// TIA Portal V18 program export: 1 tag tables, 0 data types, 4 data blocks, 9 code blocks (in call order from the OBs), 0 instance data blocks

VAR_GLOBAL   // PLC tag table "PLC_Tags"
   Nut_Khoi_Dong AT %I0.0 : Bool;   // Nút khởi động vật lý
   Nut_Khoi_Dong_HMI AT %M110.0 : Bool;   // Tín hiệu mô phỏng/HMI song song cho Nút khởi động vật lý
   Nut_Khoi_Dong_HMI_Gated AT %M320.0 : Bool;   // Tín hiệu HMI đã qua xử lý chế độ cho Nút khởi động vật lý
   Nut_Khoi_Dong_Eff AT %M320.1 : Bool;   // Tín hiệu thực tế/mô phỏng hiệu dụng cho Nút khởi động vật lý
   Nut_Dung AT %I0.1 : Bool;   // Nút dừng vật lý
   Nut_Dung_HMI AT %M110.1 : Bool;   // Tín hiệu mô phỏng/HMI song song cho Nút dừng vật lý
   Nut_Dung_HMI_Gated AT %M320.2 : Bool;   // Tín hiệu HMI đã qua xử lý chế độ cho Nút dừng vật lý
   Nut_Dung_Eff AT %M320.3 : Bool;   // Tín hiệu thực tế/mô phỏng hiệu dụng cho Nút dừng vật lý
   Nut_Reset AT %I0.2 : Bool;   // Nút reset lỗi vật lý
   Nut_Reset_HMI AT %M110.2 : Bool;   // Tín hiệu mô phỏng/HMI song song cho Nút reset lỗi vật lý
   Nut_Reset_HMI_Gated AT %M320.4 : Bool;   // Tín hiệu HMI đã qua xử lý chế độ cho Nút reset lỗi vật lý
   Nut_Reset_Eff AT %M320.5 : Bool;   // Tín hiệu thực tế/mô phỏng hiệu dụng cho Nút reset lỗi vật lý
   Nut_EStop AT %I0.3 : Bool;   // Nút dừng khẩn vật lý
   Nut_EStop_HMI AT %M110.3 : Bool;   // Tín hiệu mô phỏng/HMI song song cho Nút dừng khẩn vật lý
   Nut_EStop_HMI_Gated AT %M320.6 : Bool;   // Tín hiệu HMI đã qua xử lý chế độ cho Nút dừng khẩn vật lý
   Nut_EStop_Eff AT %M320.7 : Bool;   // Tín hiệu thực tế/mô phỏng hiệu dụng cho Nút dừng khẩn vật lý
   FT3200_Bon1 AT %ID100 : Real;   // Cảm biến lưu lượng nước dosing vào Bồn 1
   FT3200_Bon1_HMI AT %MD700 : Real;   // Giá trị mô phỏng/HMI song song cho Cảm biến lưu lượng nước dosing vào Bồn 1
   FT3200_Bon1_Use_HMI AT %M420.0 : Bool;   // Chọn chế độ mô phỏng HMI cho Cảm biến lưu lượng nước dosing vào Bồn 1
   FT3200_Bon1_Sim_Req AT %M321.0 : Bool;   // Yêu cầu mô phỏng cảm biến cho Cảm biến lưu lượng nước dosing vào Bồn 1
   FT3200_Bon1_Sim_Active AT %M321.1 : Bool;   // Mô phỏng cảm biến đang hoạt động cho Cảm biến lưu lượng nước dosing vào Bồn 1
   FT3200_Bon1_Eff AT %MD704 : Real;   // Giá trị thực tế/mô phỏng hiệu dụng cho Cảm biến lưu lượng nước dosing vào Bồn 1
   FQ3200_Bon1 AT %ID104 : Real;   // Bộ đếm lưu lượng tích lũy Bồn 1
   FQ3200_Bon1_HMI AT %MD708 : Real;   // Giá trị mô phỏng/HMI song song cho Bộ đếm lưu lượng tích lũy Bồn 1
   FQ3200_Bon1_Use_HMI AT %M420.1 : Bool;   // Chọn chế độ mô phỏng HMI cho Bộ đếm lưu lượng tích lũy Bồn 1
   FQ3200_Bon1_Sim_Req AT %M321.2 : Bool;   // Yêu cầu mô phỏng cảm biến cho Bộ đếm lưu lượng tích lũy Bồn 1
   FQ3200_Bon1_Sim_Active AT %M321.3 : Bool;   // Mô phỏng cảm biến đang hoạt động cho Bộ đếm lưu lượng tích lũy Bồn 1
   FQ3200_Bon1_Eff AT %MD712 : Real;   // Giá trị thực tế/mô phỏng hiệu dụng cho Bộ đếm lưu lượng tích lũy Bồn 1
   LS3202_Bon1_Cao AT %I0.4 : Bool;   // Cảm biến mức cao Bồn 1
   LS3202_Bon1_Cao_HMI AT %M110.4 : Bool;   // Tín hiệu mô phỏng/HMI song song cho Cảm biến mức cao Bồn 1
   LS3202_Bon1_Cao_HMI_Gated AT %M321.4 : Bool;   // Tín hiệu HMI đã qua xử lý chế độ cho Cảm biến mức cao Bồn 1
   LS3202_Bon1_Cao_Eff AT %M321.5 : Bool;   // Tín hiệu thực tế/mô phỏng hiệu dụng cho Cảm biến mức cao Bồn 1
   LT3203_Bon1 AT %ID108 : Real;   // Cảm biến mức liên tục Bồn 1
   LT3203_Bon1_HMI AT %MD716 : Real;   // Giá trị mô phỏng/HMI song song cho Cảm biến mức liên tục Bồn 1
   LT3203_Bon1_Use_HMI AT %M420.2 : Bool;   // Chọn chế độ mô phỏng HMI cho Cảm biến mức liên tục Bồn 1
   LT3203_Bon1_Sim_Req AT %M321.6 : Bool;   // Yêu cầu mô phỏng cảm biến cho Cảm biến mức liên tục Bồn 1
   LT3203_Bon1_Sim_Active AT %M321.7 : Bool;   // Mô phỏng cảm biến đang hoạt động cho Cảm biến mức liên tục Bồn 1
   LT3203_Bon1_Eff AT %MD720 : Real;   // Giá trị thực tế/mô phỏng hiệu dụng cho Cảm biến mức liên tục Bồn 1
   TT3204_Bon1 AT %ID112 : Real;   // Cảm biến nhiệt độ Bồn 1
   TT3204_Bon1_HMI AT %MD724 : Real;   // Giá trị mô phỏng/HMI song song cho Cảm biến nhiệt độ Bồn 1
   TT3204_Bon1_Use_HMI AT %M420.3 : Bool;   // Chọn chế độ mô phỏng HMI cho Cảm biến nhiệt độ Bồn 1
   TT3204_Bon1_Sim_Req AT %M322.0 : Bool;   // Yêu cầu mô phỏng cảm biến cho Cảm biến nhiệt độ Bồn 1
   TT3204_Bon1_Sim_Active AT %M322.1 : Bool;   // Mô phỏng cảm biến đang hoạt động cho Cảm biến nhiệt độ Bồn 1
   TT3204_Bon1_Eff AT %MD728 : Real;   // Giá trị thực tế/mô phỏng hiệu dụng cho Cảm biến nhiệt độ Bồn 1
   FT3205_Bon2 AT %ID116 : Real;   // Cảm biến lưu lượng nước dosing vào Bồn 2
   FT3205_Bon2_HMI AT %MD732 : Real;   // Giá trị mô phỏng/HMI song song cho Cảm biến lưu lượng nước dosing vào Bồn 2
   FT3205_Bon2_Use_HMI AT %M420.4 : Bool;   // Chọn chế độ mô phỏng HMI cho Cảm biến lưu lượng nước dosing vào Bồn 2
   FT3205_Bon2_Sim_Req AT %M322.2 : Bool;   // Yêu cầu mô phỏng cảm biến cho Cảm biến lưu lượng nước dosing vào Bồn 2
   FT3205_Bon2_Sim_Active AT %M322.3 : Bool;   // Mô phỏng cảm biến đang hoạt động cho Cảm biến lưu lượng nước dosing vào Bồn 2
   FT3205_Bon2_Eff AT %MD736 : Real;   // Giá trị thực tế/mô phỏng hiệu dụng cho Cảm biến lưu lượng nước dosing vào Bồn 2
   FQ3205_Bon2 AT %ID120 : Real;   // Bộ đếm lưu lượng tích lũy Bồn 2
   FQ3205_Bon2_HMI AT %MD740 : Real;   // Giá trị mô phỏng/HMI song song cho Bộ đếm lưu lượng tích lũy Bồn 2
   FQ3205_Bon2_Use_HMI AT %M420.5 : Bool;   // Chọn chế độ mô phỏng HMI cho Bộ đếm lưu lượng tích lũy Bồn 2
   FQ3205_Bon2_Sim_Req AT %M322.4 : Bool;   // Yêu cầu mô phỏng cảm biến cho Bộ đếm lưu lượng tích lũy Bồn 2
   FQ3205_Bon2_Sim_Active AT %M322.5 : Bool;   // Mô phỏng cảm biến đang hoạt động cho Bộ đếm lưu lượng tích lũy Bồn 2
   FQ3205_Bon2_Eff AT %MD744 : Real;   // Giá trị thực tế/mô phỏng hiệu dụng cho Bộ đếm lưu lượng tích lũy Bồn 2
   LT3209_Bon2 AT %ID124 : Real;   // Cảm biến mức liên tục Bồn 2
   LT3209_Bon2_HMI AT %MD748 : Real;   // Giá trị mô phỏng/HMI song song cho Cảm biến mức liên tục Bồn 2
   LT3209_Bon2_Use_HMI AT %M420.6 : Bool;   // Chọn chế độ mô phỏng HMI cho Cảm biến mức liên tục Bồn 2
   LT3209_Bon2_Sim_Req AT %M322.6 : Bool;   // Yêu cầu mô phỏng cảm biến cho Cảm biến mức liên tục Bồn 2
   LT3209_Bon2_Sim_Active AT %M322.7 : Bool;   // Mô phỏng cảm biến đang hoạt động cho Cảm biến mức liên tục Bồn 2
   LT3209_Bon2_Eff AT %MD752 : Real;   // Giá trị thực tế/mô phỏng hiệu dụng cho Cảm biến mức liên tục Bồn 2
   TT3208_Bon2 AT %ID128 : Real;   // Cảm biến nhiệt độ Bồn 2
   TT3208_Bon2_HMI AT %MD756 : Real;   // Giá trị mô phỏng/HMI song song cho Cảm biến nhiệt độ Bồn 2
   TT3208_Bon2_Use_HMI AT %M420.7 : Bool;   // Chọn chế độ mô phỏng HMI cho Cảm biến nhiệt độ Bồn 2
   TT3208_Bon2_Sim_Req AT %M323.0 : Bool;   // Yêu cầu mô phỏng cảm biến cho Cảm biến nhiệt độ Bồn 2
   TT3208_Bon2_Sim_Active AT %M323.1 : Bool;   // Mô phỏng cảm biến đang hoạt động cho Cảm biến nhiệt độ Bồn 2
   TT3208_Bon2_Eff AT %MD760 : Real;   // Giá trị thực tế/mô phỏng hiệu dụng cho Cảm biến nhiệt độ Bồn 2
   VFD_Bon2_Contactor AT %Q0.0 : Bool;   // Contactor cấp nguồn/cho phép VFD Bồn 2
   VFD_Bon2_Contactor_M AT %M220.0 : Bool;   // Tag gương phản hồi HMI cho Contactor cấp nguồn/cho phép VFD Bồn 2
   CV3201_Nuoc_Bon1 AT %QD100 : Real;   // Van tuyến tính cấp nước Bồn 1
   CV3201_Nuoc_Bon1_M AT %MD1200 : Real;   // Tag gương phản hồi HMI cho Van tuyến tính cấp nước Bồn 1
   AGTR3260_Khuay_Bon1 AT %Q0.1 : Bool;   // Động cơ khuấy Bồn 1
   AGTR3260_Khuay_Bon1_M AT %M220.1 : Bool;   // Tag gương phản hồi HMI cho Động cơ khuấy Bồn 1
   AGTR3260_Toc_Do_AO AT %QD104 : Real;   // Tín hiệu tốc độ khuấy Bồn 1
   AGTR3260_Toc_Do_AO_M AT %MD1204 : Real;   // Tag gương phản hồi HMI cho Tín hiệu tốc độ khuấy Bồn 1
   V3232_Xa_Bon1 AT %Q0.2 : Bool;   // Van xả đáy Bồn 1 số 1
   V3232_Xa_Bon1_M AT %M220.2 : Bool;   // Tag gương phản hồi HMI cho Van xả đáy Bồn 1 số 1
   V3233_Xa_Bon1 AT %Q0.3 : Bool;   // Van xả đáy Bồn 1 số 2
   V3233_Xa_Bon1_M AT %M220.3 : Bool;   // Tag gương phản hồi HMI cho Van xả đáy Bồn 1 số 2
   V3234_Xa_Bon1 AT %Q0.4 : Bool;   // Van xả đáy Bồn 1 số 3
   V3234_Xa_Bon1_M AT %M220.4 : Bool;   // Tag gương phản hồi HMI cho Van xả đáy Bồn 1 số 3
   V3235_Nuoc_Bon2 AT %Q0.5 : Bool;   // Van on/off cấp nước Bồn 2
   V3235_Nuoc_Bon2_M AT %M220.5 : Bool;   // Tag gương phản hồi HMI cho Van on/off cấp nước Bồn 2
   CV3206_Hoi_Bon2 AT %QD108 : Real;   // Van hơi/nhiệt Bồn 2 ở chế độ cho phép
   CV3206_Hoi_Bon2_M AT %MD1208 : Real;   // Tag gương phản hồi HMI cho Van hơi/nhiệt Bồn 2 ở chế độ cho phép
   VFD_Bon2_Dummy_Run_Physical AT %Q0.6 : Bool;   // Dummy RUN physical output VFD Bồn 2
   VFD_Bon2_Dummy_Run_Physical_M AT %M220.6 : Bool;   // Tag gương phản hồi HMI cho Dummy RUN physical output VFD Bồn 2
   VFD_Bon2_Dummy_Reverse_Physical AT %Q0.7 : Bool;   // Dummy Reverse physical output VFD Bồn 2
   VFD_Bon2_Dummy_Reverse_Physical_M AT %M220.7 : Bool;   // Tag gương phản hồi HMI cho Dummy Reverse physical output VFD Bồn 2
   VFD_Bon2_Dummy_Speed_Physical AT %QD112 : Real;   // Dummy Speed physical output VFD Bồn 2
   VFD_Bon2_Dummy_Speed_Physical_M AT %MD1212 : Real;   // Tag gương phản hồi HMI cho Dummy Speed physical output VFD Bồn 2
   V3237_Xa_Bon2 AT %Q1.0 : Bool;   // Van xả đáy Bồn 2 số 1
   V3237_Xa_Bon2_M AT %M221.0 : Bool;   // Tag gương phản hồi HMI cho Van xả đáy Bồn 2 số 1
   V3238_Xa_Bon2 AT %Q1.1 : Bool;   // Van xả đáy Bồn 2 số 2
   V3238_Xa_Bon2_M AT %M221.1 : Bool;   // Tag gương phản hồi HMI cho Van xả đáy Bồn 2 số 2
   V3239_Xa_Bon2 AT %Q1.2 : Bool;   // Van xả đáy Bồn 2 số 3
   V3239_Xa_Bon2_M AT %M221.2 : Bool;   // Tag gương phản hồi HMI cho Van xả đáy Bồn 2 số 3
   Pump3264_Chuyen_Nhanh1 AT %Q1.3 : Bool;   // Bơm chuyển dung dịch Nhánh 1 xuống bồn chứa
   Pump3264_Chuyen_Nhanh1_M AT %M221.3 : Bool;   // Tag gương phản hồi HMI cho Bơm chuyển dung dịch Nhánh 1 xuống bồn chứa
   LT3302_BonChua1 AT %ID164 : Real;   // Cảm biến mức liên tục Bồn chứa 01
   LT3302_BonChua1_HMI AT %MD828 : Real;   // Giá trị mô phỏng/HMI song song cho Cảm biến mức liên tục Bồn chứa 01
   LT3302_BonChua1_Use_HMI AT %M422.0 : Bool;   // Chọn chế độ mô phỏng HMI cho Cảm biến mức liên tục Bồn chứa 01
   LT3302_BonChua1_Sim_Req AT %M325.4 : Bool;   // Yêu cầu mô phỏng cảm biến cho Cảm biến mức liên tục Bồn chứa 01
   LT3302_BonChua1_Sim_Active AT %M325.5 : Bool;   // Mô phỏng cảm biến đang hoạt động cho Cảm biến mức liên tục Bồn chứa 01
   LT3302_BonChua1_Eff AT %MD832 : Real;   // Giá trị thực tế/mô phỏng hiệu dụng cho Cảm biến mức liên tục Bồn chứa 01
   TT3301_BonChua1 AT %ID168 : Real;   // Cảm biến nhiệt độ Bồn chứa 01
   TT3301_BonChua1_HMI AT %MD836 : Real;   // Giá trị mô phỏng/HMI song song cho Cảm biến nhiệt độ Bồn chứa 01
   TT3301_BonChua1_Use_HMI AT %M422.1 : Bool;   // Chọn chế độ mô phỏng HMI cho Cảm biến nhiệt độ Bồn chứa 01
   TT3301_BonChua1_Sim_Req AT %M325.6 : Bool;   // Yêu cầu mô phỏng cảm biến cho Cảm biến nhiệt độ Bồn chứa 01
   TT3301_BonChua1_Sim_Active AT %M325.7 : Bool;   // Mô phỏng cảm biến đang hoạt động cho Cảm biến nhiệt độ Bồn chứa 01
   TT3301_BonChua1_Eff AT %MD840 : Real;   // Giá trị thực tế/mô phỏng hiệu dụng cho Cảm biến nhiệt độ Bồn chứa 01
   TT3303_TraoDoiNhiet AT %ID172 : Real;   // Cảm biến nhiệt độ bộ trao đổi nhiệt
   TT3303_TraoDoiNhiet_HMI AT %MD844 : Real;   // Giá trị mô phỏng/HMI song song cho Cảm biến nhiệt độ bộ trao đổi nhiệt
   TT3303_TraoDoiNhiet_Use_HMI AT %M422.2 : Bool;   // Chọn chế độ mô phỏng HMI cho Cảm biến nhiệt độ bộ trao đổi nhiệt
   TT3303_TraoDoiNhiet_Sim_Req AT %M326.0 : Bool;   // Yêu cầu mô phỏng cảm biến cho Cảm biến nhiệt độ bộ trao đổi nhiệt
   TT3303_TraoDoiNhiet_Sim_Active AT %M326.1 : Bool;   // Mô phỏng cảm biến đang hoạt động cho Cảm biến nhiệt độ bộ trao đổi nhiệt
   TT3303_TraoDoiNhiet_Eff AT %MD848 : Real;   // Giá trị thực tế/mô phỏng hiệu dụng cho Cảm biến nhiệt độ bộ trao đổi nhiệt
   LT3307_BonChua2 AT %ID176 : Real;   // Cảm biến mức liên tục Bồn chứa 02
   LT3307_BonChua2_HMI AT %MD852 : Real;   // Giá trị mô phỏng/HMI song song cho Cảm biến mức liên tục Bồn chứa 02
   LT3307_BonChua2_Use_HMI AT %M422.3 : Bool;   // Chọn chế độ mô phỏng HMI cho Cảm biến mức liên tục Bồn chứa 02
   LT3307_BonChua2_Sim_Req AT %M326.2 : Bool;   // Yêu cầu mô phỏng cảm biến cho Cảm biến mức liên tục Bồn chứa 02
   LT3307_BonChua2_Sim_Active AT %M326.3 : Bool;   // Mô phỏng cảm biến đang hoạt động cho Cảm biến mức liên tục Bồn chứa 02
   LT3307_BonChua2_Eff AT %MD856 : Real;   // Giá trị thực tế/mô phỏng hiệu dụng cho Cảm biến mức liên tục Bồn chứa 02
   TT3306_BonChua2 AT %ID180 : Real;   // Cảm biến nhiệt độ Bồn chứa 02
   TT3306_BonChua2_HMI AT %MD860 : Real;   // Giá trị mô phỏng/HMI song song cho Cảm biến nhiệt độ Bồn chứa 02
   TT3306_BonChua2_Use_HMI AT %M422.4 : Bool;   // Chọn chế độ mô phỏng HMI cho Cảm biến nhiệt độ Bồn chứa 02
   TT3306_BonChua2_Sim_Req AT %M326.4 : Bool;   // Yêu cầu mô phỏng cảm biến cho Cảm biến nhiệt độ Bồn chứa 02
   TT3306_BonChua2_Sim_Active AT %M326.5 : Bool;   // Mô phỏng cảm biến đang hoạt động cho Cảm biến nhiệt độ Bồn chứa 02
   TT3306_BonChua2_Eff AT %MD864 : Real;   // Giá trị thực tế/mô phỏng hiệu dụng cho Cảm biến nhiệt độ Bồn chứa 02
   PI3308_Truoc_Filter AT %ID184 : Real;   // Cảm biến áp suất trước màng lọc
   PI3308_Truoc_Filter_HMI AT %MD868 : Real;   // Giá trị mô phỏng/HMI song song cho Cảm biến áp suất trước màng lọc
   PI3308_Truoc_Filter_Use_HMI AT %M422.5 : Bool;   // Chọn chế độ mô phỏng HMI cho Cảm biến áp suất trước màng lọc
   PI3308_Truoc_Filter_Sim_Req AT %M326.6 : Bool;   // Yêu cầu mô phỏng cảm biến cho Cảm biến áp suất trước màng lọc
   PI3308_Truoc_Filter_Sim_Active AT %M326.7 : Bool;   // Mô phỏng cảm biến đang hoạt động cho Cảm biến áp suất trước màng lọc
   PI3308_Truoc_Filter_Eff AT %MD872 : Real;   // Giá trị thực tế/mô phỏng hiệu dụng cho Cảm biến áp suất trước màng lọc
   FT3309_Xa_Thanh_Pham AT %ID188 : Real;   // Cảm biến lưu lượng xả thành phẩm
   FT3309_Xa_Thanh_Pham_HMI AT %MD876 : Real;   // Giá trị mô phỏng/HMI song song cho Cảm biến lưu lượng xả thành phẩm
   FT3309_Xa_Thanh_Pham_Use_HMI AT %M422.6 : Bool;   // Chọn chế độ mô phỏng HMI cho Cảm biến lưu lượng xả thành phẩm
   FT3309_Xa_Thanh_Pham_Sim_Req AT %M327.0 : Bool;   // Yêu cầu mô phỏng cảm biến cho Cảm biến lưu lượng xả thành phẩm
   FT3309_Xa_Thanh_Pham_Sim_Active AT %M327.1 : Bool;   // Mô phỏng cảm biến đang hoạt động cho Cảm biến lưu lượng xả thành phẩm
   FT3309_Xa_Thanh_Pham_Eff AT %MD880 : Real;   // Giá trị thực tế/mô phỏng hiệu dụng cho Cảm biến lưu lượng xả thành phẩm
   LSH3310_Pheu_Cao AT %I0.6 : Bool;   // Cảm biến mức cao phễu chiết rót
   LSH3310_Pheu_Cao_HMI AT %M110.6 : Bool;   // Tín hiệu mô phỏng/HMI song song cho Cảm biến mức cao phễu chiết rót
   LSH3310_Pheu_Cao_HMI_Gated AT %M327.2 : Bool;   // Tín hiệu HMI đã qua xử lý chế độ cho Cảm biến mức cao phễu chiết rót
   LSH3310_Pheu_Cao_Eff AT %M327.3 : Bool;   // Tín hiệu thực tế/mô phỏng hiệu dụng cho Cảm biến mức cao phễu chiết rót
   LSL3311_Pheu_Thap AT %I0.7 : Bool;   // Cảm biến mức thấp phễu chiết rót
   LSL3311_Pheu_Thap_HMI AT %M110.7 : Bool;   // Tín hiệu mô phỏng/HMI song song cho Cảm biến mức thấp phễu chiết rót
   LSL3311_Pheu_Thap_HMI_Gated AT %M327.4 : Bool;   // Tín hiệu HMI đã qua xử lý chế độ cho Cảm biến mức thấp phễu chiết rót
   LSL3311_Pheu_Thap_Eff AT %M327.5 : Bool;   // Tín hiệu thực tế/mô phỏng hiệu dụng cho Cảm biến mức thấp phễu chiết rót
   V3331_Xa_BonChua1 AT %Q3.0 : Bool;   // Van xả đáy Bồn chứa 01 số 1
   V3331_Xa_BonChua1_M AT %M223.0 : Bool;   // Tag gương phản hồi HMI cho Van xả đáy Bồn chứa 01 số 1
   V3332_Xa_BonChua1 AT %Q3.1 : Bool;   // Van xả đáy Bồn chứa 01 số 2
   V3332_Xa_BonChua1_M AT %M223.1 : Bool;   // Tag gương phản hồi HMI cho Van xả đáy Bồn chứa 01 số 2
   Pump3361_LuanChuyen_BonChua1 AT %Q3.2 : Bool;   // Bơm luân chuyển Bồn chứa 01
   Pump3361_LuanChuyen_BonChua1_M AT %M223.2 : Bool;   // Tag gương phản hồi HMI cho Bơm luân chuyển Bồn chứa 01
   Pump3362_Xa_BonChua1 AT %Q3.3 : Bool;   // Bơm xả Bồn chứa 01
   Pump3362_Xa_BonChua1_M AT %M223.3 : Bool;   // Tag gương phản hồi HMI cho Bơm xả Bồn chứa 01
   V3333_DieuHuong_BonChua1 AT %Q3.4 : Bool;   // Van điều hướng Bồn chứa 01 số 1
   V3333_DieuHuong_BonChua1_M AT %M223.4 : Bool;   // Tag gương phản hồi HMI cho Van điều hướng Bồn chứa 01 số 1
   V3334_DieuHuong_BonChua1 AT %Q3.5 : Bool;   // Van điều hướng Bồn chứa 01 số 2
   V3334_DieuHuong_BonChua1_M AT %M223.5 : Bool;   // Tag gương phản hồi HMI cho Van điều hướng Bồn chứa 01 số 2
   V3335_DieuHuong_BonChua1 AT %Q3.6 : Bool;   // Van điều hướng Bồn chứa 01 số 3
   V3335_DieuHuong_BonChua1_M AT %M223.6 : Bool;   // Tag gương phản hồi HMI cho Van điều hướng Bồn chứa 01 số 3
   CV3304_Nuoc_Lam_Mat AT %QD132 : Real;   // Van tuyến tính nước làm mát
   CV3304_Nuoc_Lam_Mat_M AT %MD1232 : Real;   // Tag gương phản hồi HMI cho Van tuyến tính nước làm mát
   V3338_Xa_BonChua2 AT %Q3.7 : Bool;   // Van xả đáy Bồn chứa 02 số 1
   V3338_Xa_BonChua2_M AT %M223.7 : Bool;   // Tag gương phản hồi HMI cho Van xả đáy Bồn chứa 02 số 1
   V3339_Xa_BonChua2 AT %Q4.0 : Bool;   // Van xả đáy Bồn chứa 02 số 2
   V3339_Xa_BonChua2_M AT %M224.0 : Bool;   // Tag gương phản hồi HMI cho Van xả đáy Bồn chứa 02 số 2
   Pump3364_Filter AT %Q4.1 : Bool;   // Bơm qua màng lọc CCP số 1
   Pump3364_Filter_M AT %M224.1 : Bool;   // Tag gương phản hồi HMI cho Bơm qua màng lọc CCP số 1
   Pump3365_Filter AT %Q4.2 : Bool;   // Bơm qua màng lọc CCP số 2
   Pump3365_Filter_M AT %M224.2 : Bool;   // Tag gương phản hồi HMI cho Bơm qua màng lọc CCP số 2
   V3340_Duong_Filter AT %Q4.3 : Bool;   // Van đường ống Filter số 1
   V3340_Duong_Filter_M AT %M224.3 : Bool;   // Tag gương phản hồi HMI cho Van đường ống Filter số 1
   V3341_Duong_Filter AT %Q4.4 : Bool;   // Van đường ống Filter số 2
   V3341_Duong_Filter_M AT %M224.4 : Bool;   // Tag gương phản hồi HMI cho Van đường ống Filter số 2
   CV_Filler_Cap_Dich AT %QD136 : Real;   // Van tuyến tính cấp dịch xuống phễu chiết rót
   CV_Filler_Cap_Dich_M AT %MD1236 : Real;   // Tag gương phản hồi HMI cho Van tuyến tính cấp dịch xuống phễu chiết rót
   Coi_Bao_Dong AT %Q4.5 : Bool;   // Còi báo động chung
   Coi_Bao_Dong_M AT %M224.5 : Bool;   // Tag gương phản hồi HMI cho Còi báo động chung
   HMI_Operator_Login AT %M422.7 : Bool;   // Đăng nhập quyền Operator
   HMI_Engineer_Login AT %M423.0 : Bool;   // Đăng nhập quyền Engineer
   HMI_Admin_Login AT %M423.1 : Bool;   // Đăng nhập quyền Admin
   HMI_Che_Do_Manual AT %M423.2 : Bool;   // Cho phép điều khiển tay từng thiết bị
   HMI_Ack_Alarm AT %M423.3 : Bool;   // Xác nhận cảnh báo
   HMI_Reset_Alarm AT %M423.4 : Bool;   // Reset alarm bằng HMI
   Gia_Lap_Mat_Ket_Noi_HMI AT %M423.5 : Bool;   // Nút giả lập mất kết nối PLC
   HMI_User_Level AT %MW520 : Int;   // Mức quyền hiện tại: 1 Operator, 2 Engineer, 3 Admin
   HMI_Cho_Phep_Sua_Thong_So AT %M327.6 : Bool;   // Cờ cho phép sửa công thức và PID
   HMI_Alarm_Status AT %MW522 : Int;   // Mã cảnh báo tổng hợp cho WinCC TextList
   HMI_AnToan_Status AT %MW524 : Int;   // Mã chẩn đoán an toàn ưu tiên
   PLC1_Auto_Enable AT %M327.7 : Bool;   // Cho phép chạy Auto Nhánh 1 Bồn 1-2
   PLC1_EStop_Latch AT %M328.0 : Bool;   // Chốt dừng khẩn HMI/SCADA Nhánh 1 Bồn 1-2
   PLC1_Loi_Tong AT %M328.1 : Bool;   // Lỗi tổng khóa Auto Nhánh 1 Bồn 1-2
   PLC1_Loi_Dry_Run AT %M328.2 : Bool;   // Lỗi chạy khô bơm Nhánh 1 Bồn 1-2
   PLC1_Loi_Dosing AT %M328.3 : Bool;   // Lỗi quá thời gian dosing Nhánh 1 Bồn 1-2
   PLC1_Loi_Truyen_Thong AT %M328.4 : Bool;   // Lỗi truyền thông mô phỏng Nhánh 1 Bồn 1-2
   PLC1_State AT %MW526 : Int;   // Mã bước chu trình Nhánh 1 Bồn 1-2
   PLC1_Step_Bon1_Dosing AT %M329.3 : Bool;   // Bồn 1 đang dosing nước
   PLC1_Step_Bon1_Tip AT %M329.4 : Bool;   // Bồn 1 đang mô phỏng tip cốt tương Nhật Bản
   PLC1_Step_Bon1_Khuay AT %M329.5 : Bool;   // Bồn 1 đang khuấy ban đầu
   PLC1_Step_Bon1_Xa AT %M329.6 : Bool;   // Bồn 1 đang xả sang Bồn 2
   PLC1_Step_Bon2_Dosing AT %M329.7 : Bool;   // Bồn 2 đang dosing bổ sung
   PLC1_Step_Bon2_Tip AT %M330.0 : Bool;   // Bồn 2 đang tip phụ gia
   PLC1_Step_Bon2_Khuay_Thuan AT %M330.1 : Bool;   // Bồn 2 khuấy chiều thuận
   PLC1_Step_Bon2_Khuay_Nghich AT %M330.2 : Bool;   // Bồn 2 khuấy chiều ngược
   PLC1_Step_Bon2_PID AT %M330.3 : Bool;   // Bồn 2 gia nhiệt PID
   PLC1_Step_Bon2_Thanh_Trung AT %M330.4 : Bool;   // Bồn 2 giữ thời gian thanh trùng
   PLC1_Me_Nhanh1_Hoan_Thanh AT %M330.5 : Bool;   // Nhánh 1 hoàn thành và sẵn sàng xả xuống bồn chứa
   PLC1_Xa_Bon1_Xong AT %M330.6 : Bool;   // Bồn 1 đã xả hết
   PLC1_Xa_Bon2_Xong AT %M330.7 : Bool;   // Bồn 2 đã xả hết
   BonChua_Step_Nhan_Dich AT %M332.4 : Bool;   // Bồn chứa 01 đang nhận dịch từ nhánh hoàn thành
   BonChua_Step_Giai_Nhiet AT %M332.5 : Bool;   // Bồn chứa 01 đang giải nhiệt xuống 45 độ C
   BonChua_Step_Chuyen_Bon2 AT %M332.6 : Bool;   // Đang chuyển từ Bồn chứa 01 sang Bồn chứa 02
   BonChua_Step_Loc_Chiet AT %M332.7 : Bool;   // Đang lọc CCP và chiết rót
   BonChua_Me_Hoan_Thanh AT %M333.0 : Bool;   // Hoàn thành một mẻ sản xuất chung
   BonChua_State AT %MW530 : Int;   // Mã bước cụm bồn chứa và lọc thành phẩm
   BonChua_Owner_Nhanh1 AT %M333.1 : Bool;   // Mức ưu tiên Nhánh 1 sở hữu bồn chứa
   BonChua_Owner_Nhanh2 AT %M333.2 : Bool;   // Mức ưu tiên Nhánh 2 sở hữu bồn chứa
   PLC2_Me_Nhanh2_Hoan_Thanh_Nhan AT %M333.4 : Bool;   // Cờ PLC1 nhận trạng thái hoàn thành từ PLC2
   PLC2_Me_Nhanh2_Hoan_Thanh_Nhan_HMI AT %M111.0 : Bool;   // Tín hiệu mô phỏng/HMI song song cho cờ PLC1 nhận trạng thái hoàn thành từ PLC2
   PLC2_Xa_Bon4_Xong_Nhan AT %M333.5 : Bool;   // Cờ PLC1 nhận trạng thái xả xong Bồn 4 từ PLC2
   Pump3265_Chuyen_Nhanh2_Cmd AT %M333.6 : Bool;   // Lệnh chạy bơm chuyển Nhánh 2 gửi sang PLC2
   Pump3265_Chuyen_Nhanh2_Cmd_M AT %M224.7 : Bool;   // Tag gương phản hồi HMI cho lệnh chạy bơm chuyển Nhánh 2 gửi sang PLC2
   PID_Bon4_SP_Recv AT %MD884 : Real;   // PID Bồn 4 Setpoint nhận từ PLC2
   PID_Bon4_PV_Recv AT %MD888 : Real;   // PID Bồn 4 Process Value nhận từ PLC2
   PID_Bon4_CV_Recv AT %MD892 : Real;   // PID Bồn 4 Control Value nhận từ PLC2
   PLC2_State_Recv AT %MW532 : Int;   // Trạng thái hoạt động PLC2 nhận từ PLC2
   PLC2_Loi_Tong_Recv AT %M334.0 : Bool;   // Cờ lỗi tổng PLC2 nhận từ PLC2
   VFD_Bon2_iStep AT %MW60 : Int;   // Bước quét tuần tự Modbus VFD Bồn 2
   VFD_Bon2_iStep_Reset AT %M335.5 : Bool;   // Cờ reset bộ đếm bước Modbus VFD Bồn 2
   VFD_Bon2_Step0_Req AT %M335.6 : Bool;   // Yêu cầu bước 0 Modbus VFD Bồn 2
   VFD_Bon2_Step1_Req AT %M335.7 : Bool;   // Yêu cầu bước 1 Modbus VFD Bồn 2
   VFD_Bon2_Step2_Req AT %M336.0 : Bool;   // Yêu cầu bước 2 Modbus VFD Bồn 2
   VFD_Bon2_Step3_Req AT %M336.1 : Bool;   // Yêu cầu bước 3 Modbus VFD Bồn 2
   VFD_Bon2_MB_ControlWord AT %MW40 : Word;   // Control Word gửi VFD Bồn 2
   VFD_Bon2_MB_FreqSetpoint AT %MW42 : Int;   // Frequency Setpoint gửi VFD Bồn 2
   VFD_Bon2_MB_StatusWord AT %MW44 : Word;   // Status Word đọc từ VFD Bồn 2
   VFD_Bon2_MB_FreqActual AT %MW46 : Int;   // Actual Speed đọc từ VFD Bồn 2
   VFD_Bon2_MB_Error AT %M50.0 : Bool;   // Lỗi Modbus Master VFD Bồn 2
   VFD_Bon2_MB_Busy AT %M50.1 : Bool;   // Modbus Master Busy VFD Bồn 2
   VFD_Bon2_MB_Done AT %M50.2 : Bool;   // Modbus Master Done VFD Bồn 2
   VFD_Bon2_MB_Status AT %MW52 : Word;   // Trạng thái Modbus Master VFD Bồn 2
   VFD_Bon2_MBCL_Done AT %M51.0 : Bool;   // Modbus Comm Load Done VFD Bồn 2
   VFD_Bon2_MBCL_Error AT %M51.1 : Bool;   // Modbus Comm Load Error VFD Bồn 2
   VFD_Bon2_MBCL_Status AT %MW54 : Word;   // Trạng thái Modbus Comm Load VFD Bồn 2
   VFD_Bon2_Freq_Temp AT %MD70 : Real;   // Biến tạm tần số VFD Bồn 2
   VFD_Bon2_Actual_Speed_Feedback AT %MD74 : Real;   // Phản hồi tốc độ thực tế VFD Bồn 2
   VFD_Bon2_Actual_Speed_Feedback_M AT %MD1240 : Real;   // Tag gương phản hồi HMI tốc độ thực tế VFD Bồn 2
   MB_TCP_iStep AT %MW80 : Int;   // Modbus TCP Client step
   MB_TCP_REQ AT %M82.0 : Bool;   // Modbus TCP Client Request
   MB_TCP_DONE AT %M82.2 : Bool;   // Modbus TCP Client Transaction Done
   MB_TCP_ERROR AT %M82.3 : Bool;   // Modbus TCP Client Transaction Error
   MB_TCP_BUSY AT %M82.6 : Bool;   // Modbus TCP Client Transaction Busy
   MB_TCP_STATUS AT %MW86 : Word;   // Modbus TCP Client Status
   MB_TCP_Mode AT %MB88 : USInt;   // Modbus TCP Client Mode
   MB_TCP_DataAddr AT %MD90 : UDInt;   // Modbus TCP Client Data Address
   MB_TCP_DataLen AT %MW94 : UInt;   // Modbus TCP Client Data Length
   Nut_Khoi_Dong_Eff_Old AT %M83.0 : Bool;   // Old value of Start button
   Nut_Khoi_Dong_Eff_Edge AT %M83.6 : Bool;   // Start command edge detected
   Nut_Dung_Eff_Old AT %M83.1 : Bool;   // Old value of Stop button
   Nut_Dung_Eff_Edge AT %M83.7 : Bool;   // Stop command edge detected
   Nut_Reset_Eff_Old AT %M83.2 : Bool;   // Old value of Reset button
   Nut_Reset_Eff_Edge AT %M84.0 : Bool;   // Reset command edge detected
   Nut_EStop_Eff_Old AT %M83.3 : Bool;   // Old value of EStop button
   Nut_EStop_Eff_Edge AT %M84.1 : Bool;   // EStop command edge detected
   Pump3265_Chuyen_Nhanh2_Cmd_Old AT %M83.4 : Bool;   // Old value of Transfer command
   Pump3265_Chuyen_Nhanh2_Cmd_Edge AT %M84.2 : Bool;   // Transfer command edge detected
   PLC1_Load_Default_Cmd_Old AT %M83.5 : Bool;   // Old value of Load Recipe command
   PLC1_Load_Default_Cmd_Edge AT %M84.3 : Bool;   // Load Recipe command edge detected
   MB_TCP_Any_Cmd_Edge AT %M84.4 : Bool;   // Any handshake command edge detected
   PLC1_Tip_Bon1_Xong_HMI AT %M423.6 : Bool;   // Nút mô phỏng tip Bồn 1 đã hoàn tất
   PLC1_Khuay_Bon1_Xong_HMI AT %M423.7 : Bool;   // Nút mô phỏng hết thời gian khuấy Bồn 1
   PLC1_Tip_Bon2_Xong_HMI AT %M424.0 : Bool;   // Nút mô phỏng tip Bồn 2 đã hoàn tất
   PLC1_Khuay_Thuan_Bon2_Xong_HMI AT %M424.1 : Bool;   // Nút mô phỏng hết thời gian khuấy thuận Bồn 2
   PLC1_Khuay_Nghich_Bon2_Xong_HMI AT %M424.2 : Bool;   // Nút mô phỏng hết thời gian khuấy ngược Bồn 2
   PLC1_Thanh_Trung_Bon2_Xong_HMI AT %M424.3 : Bool;   // Nút mô phỏng hết thời gian thanh trùng Bồn 2
   PLC2_Tip_Bon3_Xong_HMI AT %M424.4 : Bool;   // Nút mô phỏng tip Bồn 3 đã hoàn tất
   PLC2_Khuay_Bon3_Xong_HMI AT %M424.5 : Bool;   // Nút mô phỏng hết thời gian khuấy Bồn 3
   PLC2_Tip_Bon4_Xong_HMI AT %M424.6 : Bool;   // Nút mô phỏng tip Bồn 4 đã hoàn tất
   PLC2_Khuay_Thuan_Bon4_Xong_HMI AT %M424.7 : Bool;   // Nút mô phỏng hết thời gian khuấy thuận Bồn 4
   PLC2_Khuay_Nghich_Bon4_Xong_HMI AT %M425.0 : Bool;   // Nút mô phỏng hết thời gian khuấy ngược Bồn 4
   PLC2_Thanh_Trung_Bon4_Xong_HMI AT %M425.1 : Bool;   // Nút mô phỏng hết thời gian thanh trùng Bồn 4
   BonChua_Nhan_Dich_Xong_HMI AT %M425.2 : Bool;   // Nút mô phỏng nhận dịch vào Bồn chứa 01 xong
   BonChua_Chuyen_Bon2_Xong_HMI AT %M425.3 : Bool;   // Nút mô phỏng chuyển sang Bồn chứa 02 xong
   HMI_SP_PLC1_Nuoc_Bon1 AT %MD896 : Real;   // Lượng nước dosing Bồn 1
   HMI_SP_PLC1_Nuoc_Bon2 AT %MD900 : Real;   // Lượng nước dosing bổ sung Bồn 2
   HMI_SP_PLC1_Toc_Do_Bon1 AT %MD904 : Real;   // Tốc độ khuấy Bồn 1
   HMI_SP_PLC1_Toc_Do_Bon2_Main AT %MD908 : Real;   // Tốc độ khuấy chính Bồn 2
   HMI_SP_PLC1_Nhiet_Do_Bon2 AT %MD912 : Real;   // Setpoint nhiệt/PID Bồn 2
   HMI_SP_PLC2_Nuoc_Bon3 AT %MD916 : Real;   // Lượng nước dosing Bồn 3
   HMI_SP_PLC2_Nuoc_Bon4 AT %MD920 : Real;   // Lượng nước dosing bổ sung Bồn 4
   HMI_SP_PLC2_Toc_Do_Bon3 AT %MD924 : Real;   // Tốc độ khuấy Bồn 3
   HMI_SP_PLC2_Toc_Do_Bon4_Main AT %MD928 : Real;   // Tốc độ khuấy chính Bồn 4
   HMI_SP_PLC2_Nhiet_Do_Bon4 AT %MD932 : Real;   // Setpoint nhiệt/PID mô phỏng Bồn 4
   HMI_SP_BonChua1_Nhiet_Giai_Nhiet AT %MD936 : Real;   // Nhiệt độ giải nhiệt đích Bồn chứa 01
   HMI_SP_Loc_Ap_Suat_Max AT %MD940 : Real;   // Ngưỡng áp suất cao trước màng lọc
   HMI_SP_Time_Khuay_Bon1 AT %MD944 : Time;   // Thời gian khuấy Bồn 1
   HMI_SP_Time_Khuay_Bon3 AT %MD948 : Time;   // Thời gian khuấy Bồn 3
   HMI_SP_Time_Fwd AT %MD952 : Time;   // Thời gian khuấy chiều thuận
   HMI_SP_Time_Rev AT %MD956 : Time;   // Thời gian khuấy chiều ngược
   HMI_SP_Time_Sterilize AT %MD960 : Time;   // Thời gian giữ nhiệt thanh trùng
   PLC1_Khuay_Bon1_Xong AT %M336.2 : Bool;   // Trạng thái tự động xong khuấy Bồn 1
   PLC1_Khuay_Thuan_Bon2_Xong AT %M336.3 : Bool;   // Trạng thái tự động xong khuấy thuận Bồn 2
   PLC1_Khuay_Nghich_Bon2_Xong AT %M336.4 : Bool;   // Trạng thái tự động xong khuấy ngược Bồn 2
   PLC1_Thanh_Trung_Bon2_Xong AT %M336.5 : Bool;   // Trạng thái tự động xong thanh trùng Bồn 2
   PLC2_Khuay_Bon3_Xong AT %M336.6 : Bool;   // Trạng thái tự động xong khuấy Bồn 3
   PLC2_Khuay_Thuan_Bon4_Xong AT %M336.7 : Bool;   // Trạng thái tự động xong khuấy thuận Bồn 4
   PLC2_Khuay_Nghich_Bon4_Xong AT %M337.0 : Bool;   // Trạng thái tự động xong khuấy ngược Bồn 4
   PLC2_Thanh_Trung_Bon4_Xong AT %M337.1 : Bool;   // Trạng thái tự động xong thanh trùng Bồn 4
   PLC1_Tip_Bon1_Auto_Done AT %M337.2 : Bool;   // Trạng thái tự động xong tip Bồn 1
   PLC1_Tip_Bon2_Auto_Done AT %M337.3 : Bool;   // Trạng thái tự động xong tip Bồn 2
   PLC2_Tip_Bon3_Auto_Done AT %M337.4 : Bool;   // Trạng thái tự động xong tip Bồn 3
   PLC2_Tip_Bon4_Auto_Done AT %M337.5 : Bool;   // Trạng thái tự động xong tip Bồn 4
   PLC1_Start_Edge_Old AT %M337.6 : Bool;   // Cờ nhớ cạnh lên nút Start PLC1
   PLC1_Start_Edge_Edge AT %M337.7 : Bool;   // Xung cạnh lên nút Start PLC1
   PLC2_Start_Edge_Old AT %M338.0 : Bool;   // Cờ nhớ cạnh lên nút Start PLC2
   PLC2_Start_Edge_Edge AT %M338.1 : Bool;   // Xung cạnh lên nút Start PLC2
   PID_Bon2_Enable AT %M338.2 : Bool;   // Cho phép PID Bồn 2
   PID_Bon2_ManualEnable AT %M338.3 : Bool;   // Chế độ manual PID Bồn 2
   PID_Bon2_Error AT %M338.4 : Bool;   // Lỗi khối PID Bồn 2
   PID_Bon2_Reset_Eff AT %M338.5 : Bool;   // Reset hiệu dụng PID Bồn 2
   PID_Bon4_Enable AT %M338.6 : Bool;   // Cho phép PID mô phỏng Bồn 4
   PID_Bon4_ManualEnable AT %M338.7 : Bool;   // Chế độ manual PID Bồn 4
   PID_Bon4_Error AT %M339.0 : Bool;   // Lỗi khối PID Bồn 4
   PID_Bon4_Reset_Eff AT %M339.1 : Bool;   // Reset hiệu dụng PID Bồn 4
   PID_Bon2_ErrorBits AT %MD964 : DWord;   // Mã lỗi DWORD PID Bồn 2
   PID_Bon4_ErrorBits AT %MD968 : DWord;   // Mã lỗi DWORD PID Bồn 4
   PID_Bon2_SP AT %MD972 : Real;   // Setpoint đưa vào PID Bồn 2
   PID_Bon2_Err AT %MD976 : Real;   // Sai lệch PID Bồn 2 = SP - PV
   PID_Bon2_CV AT %MD980 : Real;   // Giá trị điều khiển PID Bồn 2
   PID_Bon2_ManualValue AT %MD984 : Real;   // Giá trị manual PID Bồn 2
   PID_Bon4_SP AT %MD988 : Real;   // Setpoint đưa vào PID mô phỏng Bồn 4
   PID_Bon4_Err AT %MD992 : Real;   // Sai lệch PID mô phỏng Bồn 4 = SP - PV
   PID_Bon4_CV AT %MD996 : Real;   // Giá trị điều khiển PID mô phỏng Bồn 4
   PID_Bon4_ManualValue AT %MD1000 : Real;   // Giá trị manual PID Bồn 4
   TT3219_Bon4_Sim AT %MD1004 : Real;   // Nhiệt độ mô phỏng nội bộ cho PID Bồn 4
   PID_Bon2_Temp_Inc AT %MD1008 : Real;   // Mức tăng nhiệt mô phỏng Bồn 2
   PID_Bon4_Tang_Nhiet_Buoc AT %MD1012 : Real;   // Mức tăng nhiệt mô phỏng mỗi chu kỳ OB31
   TT3219_Bon4_Target AT %MD1016 : Real;   // Nhiệt độ đích mô phỏng bồn 4
   TT3219_Bon4_Sim_Pure AT %MD1020 : Real;   // Nhiệt độ mô phỏng chưa có nhiễu bồn 4
   PID_Bon4_Temp_Val_1 AT %MD1024 : Real;   // Biến tạm mô phỏng nhiệt độ 1
   PID_Bon4_Temp_Val_2 AT %MD1028 : Real;   // Biến tạm mô phỏng nhiệt độ 2
   PID_Bon4_Sim_Counter AT %MD1032 : Real;   // Đồng hồ chu kỳ mô phỏng
   PID_Bon4_Sim_Angle AT %MD1036 : Real;   // Góc lượng giác nhiễu
   PID_Bon4_Sim_Sin AT %MD1040 : Real;   // Giá trị hình sin nhiễu
   PID_Bon4_Sim_Noise AT %MD1044 : Real;   // Giá trị nhiễu nhiệt độ
   PLC1_Tip_Bon1_Timer AT %MD1048 : Real;   // Bộ đếm thời gian mô phỏng tip bồn 1
   PLC1_Tip_Bon2_Timer AT %MD1052 : Real;   // Bộ đếm thời gian mô phỏng tip bồn 2
   PLC2_Tip_Bon3_Timer AT %MD1056 : Real;   // Bộ đếm thời gian mô phỏng tip bồn 3
   PLC2_Tip_Bon4_Timer AT %MD1060 : Real;   // Bộ đếm thời gian mô phỏng tip bồn 4
   PID_Bon2_State AT %MW534 : Int;   // Trạng thái khối PID Bồn 2
   PLC1_Stop_Active AT %M339.2 : Bool;   // Tín hiệu dừng active PLC1
   VFD_Bon2_Khuay_Active AT %M339.4 : Bool;   // Trạng thái khuấy Bồn 2 active
   VFD_Bon2_Should_Run AT %M339.5 : Bool;   // Yêu cầu chạy VFD Bồn 2
   HMI_Use_Sim_Input_PLC1 AT %M340.0 : Bool;   // Cho phép sử dụng đầu vào mô phỏng PLC1
   HMI_Use_Sim_Input_BonChua AT %M340.2 : Bool;   // Cho phép sử dụng đầu vào mô phỏng Bồn chứa
   PLC2_Me_Nhanh2_Hoan_Thanh_Nhan_Eff AT %M340.3 : Bool;   // Cờ nhận trạng thái hoàn thành Nhánh 2 hiệu dụng
   PLC2_Me_Nhanh2_Hoan_Thanh_Nhan_HMI_Gated AT %M340.5 : Bool;   // Cờ nhận trạng thái hoàn thành Nhánh 2 HMI gated
   PLC1_SP_Valid AT %M340.7 : Bool;   // Setpoint PLC1 hợp lệ
   BonChua_SP_Valid AT %M341.1 : Bool;   // Setpoint Bồn chứa hợp lệ
   PLC1_Loi_Setpoint AT %M341.2 : Bool;   // Lỗi Setpoint PLC1
   BonChua_Loi_Setpoint AT %M341.4 : Bool;   // Lỗi Setpoint Bồn chứa
   Init_Defaults_Done_PLC1 AT %M341.5 : Bool;   // Khởi tạo Setpoint mặc định PLC1 hoàn tất
   Init_Defaults_Done_BonChua AT %M341.7 : Bool;   // Khởi tạo Setpoint mặc định Bồn chứa hoàn tất
   Init_Trigger_PLC1 AT %M342.0 : Bool;   // Cờ kích hoạt nạp recipe mặc định PLC1
   Init_Trigger_BonChua AT %M342.2 : Bool;   // Cờ kích hoạt nạp recipe mặc định Bồn chứa
   HMI_Load_Default_Recipe AT %M342.3 : Bool;   // Yêu cầu nạp lại Recipe mặc định từ HMI
   PLC1_Load_Default_Cmd AT %M342.4 : Bool;   // Lệnh nạp recipe mặc định gửi sang PLC2
   PLC1_Load_Default_Cmd_M AT %M225.0 : Bool;   // Tag gương phản hồi HMI cho lệnh nạp recipe mặc định PLC1
   PLC1_Load_Default_Done_Nhan AT %M343.1 : Bool;   // Nhận báo nạp recipe xong từ PLC2
   PLC1_Load_Default_Done_Nhan_HMI AT %M111.7 : Bool;   // Tín hiệu mô phỏng/HMI cho nhận báo nạp recipe xong
   PLC1_Load_Default_Done_Nhan_HMI_Gated AT %M343.2 : Bool;   // Tín hiệu nhận báo nạp recipe xong HMI gated
   PLC1_Load_Default_Done_Nhan_Eff AT %M343.3 : Bool;   // Tín hiệu nhận báo nạp recipe xong hiệu dụng
   HMI_Sim_Mode AT %M343.4 : Bool;   // Cho phép toàn bộ tín hiệu mô phỏng HMI tác động vào input hiệu dụng
   HMI_Run_Enable AT %M343.5 : Bool;   // Cho phép vận hành từ HMI ở chế độ thật
   System_Mode_Real AT %M343.6 : Bool;   // Hệ thống đang hoạt động ở chế độ thực tế
   System_Mode_Sim AT %M343.7 : Bool;   // Hệ thống đang hoạt động ở chế độ mô phỏng
   HMI_Sim_Active_Warning AT %M344.0 : Bool;   // Cảnh báo chế độ mô phỏng HMI đang hoạt động
   PID_Bon2_Kp_HMI AT %MD1064 : Real;   // HMI parameter for Kp PID Bồn 2
   PID_Bon2_Ti_HMI AT %MD1068 : Real;   // HMI parameter for Ti PID Bồn 2
   BonChua_Nhan_Dich_Xong_Nhanh1 AT %M344.1 : Bool;   // Nhận dịch xong từ Nhánh 1
   BonChua_Nhan_Dich_Xong_Nhanh2 AT %M344.2 : Bool;   // Nhận dịch xong từ Nhánh 2
   Clock_1Hz_Last AT %M344.3 : Bool;   // Trạng thái Clock 1Hz chu kỳ trước
   Clock_1Hz_Edge AT %M344.4 : Bool;   // Xung cạnh lên của Clock 1Hz
   PLC2_Heartbeat_Last AT %MW540 : Int;   // Heartbeat PLC2 chu kỳ trước
   PLC2_Heartbeat_Changed AT %M344.7 : Bool;   // Cờ heartbeat PLC2 thay đổi
   PLC1_Heartbeat_Timeout AT %M345.0 : Bool;   // Lỗi timeout heartbeat PLC2
   VFD_Bon2_MB_Req AT %M345.1 : Bool;   // REQ cho VFD Modbus
   VFD_Bon2_MB_Mode AT %MB500 : USInt;   // MODE cho VFD Modbus
   VFD_Bon2_MB_DataAddr AT %MD504 : UDInt;   // DATA_ADDR cho VFD Modbus
   VFD_Bon2_MB_DataLen AT %MW508 : UInt;   // DATA_LEN cho VFD Modbus
   VFD_Bon2_MB_DataBuffer AT %MW510 : Word;   // Buffer dữ liệu cho VFD Modbus
   HMI_Anim_Bon1_Frame AT %MW542 : Int;   // Khung hình animation cánh khuấy Bồn 1 (0..7)
   HMI_Anim_Bon2_Frame AT %MW544 : Int;   // Khung hình animation cánh khuấy Bồn 2 (0..7)
   HMI_Anim_Bon1_MucDich AT %MW550 : Int;   // Hình trạng thái mức dịch Bồn 1 (0..2)
   HMI_Anim_Bon2_MucDich AT %MW552 : Int;   // Hình trạng thái mức dịch Bồn 2 (0..2)
   HMI_Anim_BonChua1_MucDich AT %MW554 : Int;   // Hình trạng thái mức dịch Bồn chứa 1 (0..2)
   HMI_Anim_BonChua2_MucDich AT %MW556 : Int;   // Hình trạng thái mức dịch Bồn chứa 2 (0..2)
   V3230_Nuoc_Bon1 AT %M345.2 : Bool;   // Van nước Bồn 1 (virtual)
   V3230_Nuoc_Bon1_M AT %M345.3 : Bool;   // Tag gương phản hồi HMI cho Van nước Bồn 1
   VFD_Bon2_Run AT %M345.4 : Bool;   // Lệnh chạy VFD Bồn 2 (virtual)
   VFD_Bon2_Run_M AT %M345.5 : Bool;   // Tag gương phản hồi HMI cho Lệnh chạy VFD Bồn 2
   VFD_Bon2_Dao_Chieu AT %M345.6 : Bool;   // Lệnh đảo chiều VFD Bồn 2 (virtual)
   VFD_Bon2_Dao_Chieu_M AT %M345.7 : Bool;   // Tag gương phản hồi HMI cho Lệnh đảo chiều VFD Bồn 2
   VFD_Bon2_Toc_Do_AO AT %MD1080 : Real;   // Tốc độ đặt VFD Bồn 2 (virtual)
   VFD_Bon2_Toc_Do_AO_M AT %MD1084 : Real;   // Tag gương phản hồi HMI cho Tốc độ đặt VFD Bồn 2
   VFD_Bon2_Contactor_Delay_Done AT %M346.0 : Bool;   // Trễ đóng contactor VFD Bồn 2 hoàn tất
   PLC1_Manual_Mode_Active AT %M346.1 : Bool;   // Cờ báo chế độ điều khiển tay PLC1 hoạt động
   BonChua1_Xa_Xong AT %M346.2 : Bool;   // Cụm bồn chứa - Bồn chứa 01 đã xả hết hoàn toàn
   BonChua2_Xa_Xong AT %M346.3 : Bool;   // Cụm bồn chứa - Bồn chứa 02 đã xả hết hoàn toàn
   V3230_Nuoc_Bon1_Man AT %M346.4 : Bool;   // Lệnh điều khiển tay van nước Bồn 1
   CV3201_Nuoc_Bon1_Man AT %MD1088 : Real;   // Giá trị mở tay van tuyến tính nước Bồn 1
   AGTR3260_Khuay_Bon1_Man AT %M346.5 : Bool;   // Lệnh điều khiển tay động cơ khuấy Bồn 1
   AGTR3260_Toc_Do_AO_Man AT %MD1092 : Real;   // Giá trị đặt tốc độ tay động cơ khuấy Bồn 1
   V3232_Xa_Bon1_Man AT %M346.6 : Bool;   // Lệnh điều khiển tay van xả đáy Bồn 1 số 1
   V3233_Xa_Bon1_Man AT %M346.7 : Bool;   // Lệnh điều khiển tay van xả đáy Bồn 1 số 2
   V3234_Xa_Bon1_Man AT %M347.0 : Bool;   // Lệnh điều khiển tay van xả đáy Bồn 1 số 3
   V3235_Nuoc_Bon2_Man AT %M347.1 : Bool;   // Lệnh điều khiển tay van nước Bồn 2
   CV3206_Hoi_Bon2_Man AT %MD1096 : Real;   // Giá trị mở tay van tuyến tính hơi Bồn 2
   VFD_Bon2_Run_Man AT %M347.2 : Bool;   // Lệnh điều khiển tay chạy VFD Bồn 2
   VFD_Bon2_Dao_Chieu_Man AT %M347.3 : Bool;   // Lệnh điều khiển tay đảo chiều VFD Bồn 2
   VFD_Bon2_Toc_Do_AO_Man AT %MD1100 : Real;   // Giá trị đặt tốc độ tay VFD Bồn 2
   V3237_Xa_Bon2_Man AT %M347.4 : Bool;   // Lệnh điều khiển tay van xả đáy Bồn 2 số 1
   V3238_Xa_Bon2_Man AT %M347.5 : Bool;   // Lệnh điều khiển tay van xả đáy Bồn 2 số 2
   V3239_Xa_Bon2_Man AT %M347.6 : Bool;   // Lệnh điều khiển tay van xả đáy Bồn 2 số 3
   Pump3264_Chuyen_Nhanh1_Man AT %M347.7 : Bool;   // Lệnh điều khiển tay bơm chuyển Nhánh 1
   V3331_Xa_BonChua1_Man AT %M348.0 : Bool;   // Lệnh điều khiển tay van xả đáy Bồn chứa 1 số 1
   V3332_Xa_BonChua1_Man AT %M348.1 : Bool;   // Lệnh điều khiển tay van xả đáy Bồn chứa 1 số 2
   Pump3361_LuanChuyen_BonChua1_Man AT %M348.2 : Bool;   // Lệnh điều khiển tay bơm luân chuyển Bồn chứa 1
   Pump3362_Xa_BonChua1_Man AT %M348.3 : Bool;   // Lệnh điều khiển tay bơm xả Bồn chứa 1
   V3333_DieuHuong_BonChua1_Man AT %M348.4 : Bool;   // Lệnh điều khiển tay van điều hướng Bồn chứa 1 số 1
   V3334_DieuHuong_BonChua1_Man AT %M348.5 : Bool;   // Lệnh điều khiển tay van điều hướng Bồn chứa 1 số 2
   V3335_DieuHuong_BonChua1_Man AT %M348.6 : Bool;   // Lệnh điều khiển tay van điều hướng Bồn chứa 1 số 3
   CV3304_Nuoc_Lam_Mat_Man AT %MD1104 : Real;   // Giá trị mở tay van nước làm mát
   V3338_Xa_BonChua2_Man AT %M348.7 : Bool;   // Lệnh điều khiển tay van xả đáy Bồn chứa 2 số 1
   V3339_Xa_BonChua2_Man AT %M349.0 : Bool;   // Lệnh điều khiển tay van xả đáy Bồn chứa 2 số 2
   Pump3364_Filter_Man AT %M349.1 : Bool;   // Lệnh điều khiển tay bơm qua lọc CCP 1
   Pump3365_Filter_Man AT %M349.2 : Bool;   // Lệnh điều khiển tay bơm qua lọc CCP 2
   V3340_Duong_Filter_Man AT %M349.3 : Bool;   // Lệnh điều khiển tay van đường Filter 1
   V3341_Duong_Filter_Man AT %M349.4 : Bool;   // Lệnh điều khiển tay van đường Filter 2
   CV_Filler_Cap_Dich_Man AT %MD1108 : Real;   // Giá trị mở tay van cấp dịch chiết rót
   HMI_Che_Do_Thi AT %MW562 : Int;   // Chế độ thi: 0=Tự động hóa (PID→Van hơi CV3206), 1=Đấu nối (PID→VFD Bồn 2 thật)
   PID_Bon2_PV_Eff AT %MD1128 : Real;   // PV hiệu dụng cho PID Bồn 2: nhiệt độ (Mode 0) hoặc tốc độ VFD (Mode 1)
   PID_Bon2_Enable_Eff AT %M351.2 : Bool;   // Enable hiệu dụng cho PID Bồn 2: theo State (Mode 0) hoặc HMI độc lập (Mode 1)
   HMI_PID_Bon2_Dau_Noi_Enable AT %M351.3 : Bool;   // HMI bật PID Bồn 2 khi Đấu nối - độc lập với State machine
   VFD_Bon2_Run_Cmd AT %M351.4 : Bool;   // Lệnh chạy VFD Bồn 2 nội bộ (chưa qua safety gate)
   VFD_Bon2_Dao_Chieu_Cmd AT %M351.5 : Bool;   // Lệnh đảo chiều VFD Bồn 2 nội bộ (chưa qua safety gate)
   VFD_Bon2_Toc_Do_Cmd AT %MD1132 : Real;   // Setpoint tốc độ VFD Bồn 2 nội bộ (chưa qua safety gate)
   HMI_VFD_Bon2_Comm_Enable AT %M351.6 : Bool;   // HMI cho phép giao tiếp Modbus RS-485 với VFD Bồn 2
   HMI_VFD_Bon2_Real_Enable AT %M351.7 : Bool;   // HMI xác nhận cho phép xuất lệnh ra VFD vật lý Bồn 2
   VFD_Bon2_Comm_Active AT %M352.0 : Bool;   // PLC tính: Modbus RS-485 VFD Bồn 2 đang active
   VFD_Bon2_Real_Active AT %M352.1 : Bool;   // PLC tính: đủ điều kiện an toàn để xuất physical outputs VFD Bồn 2
   VFD_Bon2_Run_Safe AT %M352.2 : Bool;   // Lệnh chạy VFD Bồn 2 đã qua safety gate
   VFD_Bon2_Comm_Active_Last AT %M352.3 : Bool;   // Trạng thái VFD_Bon2_Comm_Active chu kỳ trước (rising edge)
   VFD_Bon2_MBCL_Trigger AT %M352.4 : Bool;   // Trigger khởi tạo MB_COMM_LOAD khi Comm_Active cạnh lên
   VFD_Bon2_Comm_Ready AT %M352.5 : Bool;   // Truyền thông VFD Bồn 2 sẵn sàng (MB_COMM_LOAD done)
   VFD_Bon2_Mode_Invalid AT %M352.6 : Bool;   // Chế độ thi HMI_Che_Do_Thi không hợp lệ
   VFD_Bon2_MB_Error_Confirmed AT %M352.7 : Bool;   // Lỗi truyền thông Modbus VFD Bồn 2 đã xác nhận (sau 3 lần)
   VFD_Bon2_MB_Error_Counter AT %MW512 : Int;   // Bộ đếm lỗi truyền thông liên tiếp VFD Bồn 2
   VFD_Bon2_MB_Last_Status AT %MW514 : Word;   // Trạng thái lỗi Modbus VFD Bồn 2 cuối cùng
   VFD_Bon2_MB_Retry_Active AT %M353.0 : Bool;   // Cờ báo đang trong thời gian chờ 200ms để retry truyền thông
   VFD_Bon2_MB_Retry_Timer_Q AT %M353.1 : Bool;   // Tín hiệu ngõ ra Timer retry 200ms
   VFD_Bon2_MBCL_Active AT %M353.2 : Bool;   // Trạng thái đang thực thi khởi tạo MB_COMM_LOAD
   VFD_Bon2_MB_Error_Last AT %M353.3 : Bool;   // Trạng thái lỗi Modbus VFD Bồn 2 chu kỳ trước (phát hiện cạnh lên)
   VFD_Bon2_MB_Error_Edge AT %M353.4 : Bool;   // Xung cạnh lên phát hiện lỗi Modbus VFD Bồn 2
END_VAR

DATA_BLOCK "DB_PLC1_MB_Buffer_DB"   // DB12
TITLE = DB_PLC1_MB_Buffer_DB
{ S7_Optimized_Access := 'FALSE' }
VERSION : 0.1
// DB communication via Modbus TCP
// stored: AutoNumber false, IsOnlyStoredInLoadMemory false, IsWriteProtectedInAS false
   VAR
      Send_CmdSeq : Int;
      Send_Cmd_Start : Bool;
      Send_Cmd_Stop : Bool;
      Send_Cmd_Reset : Bool;
      Send_Cmd_EStop : Bool;
      Send_Cmd_Pump_Branch2_To_SubTanks : Bool;
      Send_Cmd_Load_Recipe : Bool;
      Send_Heartbeat : Int;
      Recv_AckSeq : Int;
      Recv_Done_Branch2 : Bool;
      Recv_Done_Recipe : Bool;
      Recv_Alarm : Bool;
      Recv_State : Int;
      Recv_PID_Bon4_SP : Real;
      Recv_PID_Bon4_PV : Real;
      Recv_PID_Bon4_CV : Real;
      Recv_Done_Discharge2 : Bool;
      Recv_Heartbeat : Int;
   END_VAR
BEGIN
END_DATA_BLOCK

DATA_BLOCK "DB_PLC1_Recv_From_PLC2_DB"   // DB10
TITLE = DB_PLC1_Recv_From_PLC2_DB
{ S7_Optimized_Access := 'FALSE' }
VERSION : 0.1
// DB communication via Modbus TCP
// stored: AutoNumber false, IsOnlyStoredInLoadMemory false, IsWriteProtectedInAS false
   VAR
      AckSeq : Int;
      Done_Branch2 : Bool;
      Done_Recipe : Bool;
      Alarm : Bool;
      State : Int;
      PID_Bon4_SP : Real;
      PID_Bon4_PV : Real;
      PID_Bon4_CV : Real;
      Done_Discharge2 : Bool;
      Heartbeat : Int;
   END_VAR
BEGIN
END_DATA_BLOCK

DATA_BLOCK "DB_PLC1_Send_To_PLC2_DB"   // DB11
TITLE = DB_PLC1_Send_To_PLC2_DB
{ S7_Optimized_Access := 'FALSE' }
VERSION : 0.1
// DB communication via Modbus TCP
// stored: AutoNumber false, IsOnlyStoredInLoadMemory false, IsWriteProtectedInAS false
   VAR
      CmdSeq : Int;
      Cmd_Start : Bool;
      Cmd_Stop : Bool;
      Cmd_Reset : Bool;
      Cmd_EStop : Bool;
      Cmd_Pump_Branch2_To_SubTanks : Bool;
      Cmd_Load_Recipe : Bool;
      Heartbeat : Int;
   END_VAR
BEGIN
END_DATA_BLOCK

DATA_BLOCK "Timers_PLC1"   // DB1
TITLE = Timers_PLC1
{ S7_Optimized_Access := 'TRUE' }
VERSION : 0.1
// Global DB containing all timers and PID instances
// stored: AutoNumber true, IsOnlyStoredInLoadMemory false, IsRetainMemResEnabled false, IsWriteProtectedInAS false, MemoryReserve 100
   VAR
      Timer_Dosing_Bon1 : IEC_TIMER;
      Timer_Tip_Bon1 : IEC_TIMER;
      Timer_Dosing_Bon2 : IEC_TIMER;
      Timer_Tip_Bon2 : IEC_TIMER;
      Timer_Khuay_Bon1 : IEC_TIMER;
      Timer_Khuay_Thuan_Bon2 : IEC_TIMER;
      Timer_Khuay_Nghich_Bon2 : IEC_TIMER;
      Timer_Thanh_Trung_Bon2 : IEC_TIMER;
      Timer_Heartbeat_PLC1 : IEC_TIMER;
      VFD_Bon2_MB_Counter : IEC_COUNTER;
      Timer_VFD_Contactor : IEC_TIMER;
      Timer_VFD_MB_Retry : IEC_TIMER;
   END_VAR
BEGIN
END_DATA_BLOCK

ORGANIZATION_BLOCK "Main"   // OB1, LAD, ProgramCycle
TITLE = "Main Program Sweep (Cycle)"
{ S7_Optimized_Access := 'TRUE' }
VERSION : 0.1
// stored: AutoNumber true, IsIECCheckEnabled false, SetENOAutomatically false
   VAR_INPUT
      Initial_Call : Bool;   // Initial call of this OB
      Remanence : Bool;   // =True, if remanent data are available
   END_VAR
BEGIN

REGION Network 1: Clock 1Hz Edge Detection
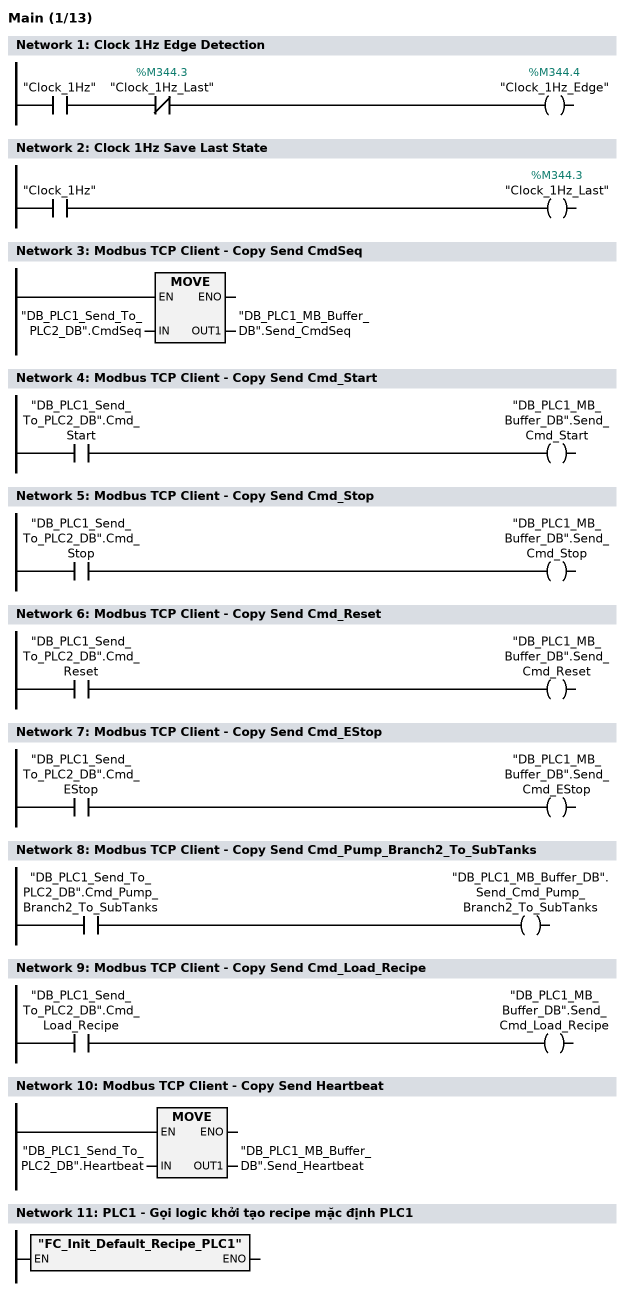
   RUNG wire#powerrail
      Contact( "Clock_1Hz" )
      I_Contact( "Clock_1Hz_Last" )
      Coil( "Clock_1Hz_Edge" )
   END_RUNG
   // the same network as SCL:
   "Clock_1Hz_Edge" := "Clock_1Hz" AND NOT "Clock_1Hz_Last";
END_REGION

REGION Network 2: Clock 1Hz Save Last State
   RUNG wire#powerrail
      Contact( "Clock_1Hz" )
      Coil( "Clock_1Hz_Last" )
   END_RUNG
   // the same network as SCL:
   "Clock_1Hz_Last" := "Clock_1Hz";
END_REGION

REGION Network 3: Modbus TCP Client - Copy Send CmdSeq
   RUNG wire#powerrail
      { S7_GenerateENO := "TRUE" } Move(in := "DB_PLC1_Send_To_PLC2_DB".CmdSeq, out1 => "DB_PLC1_MB_Buffer_DB".Send_CmdSeq)
   END_RUNG
   // the same network as SCL:
   "DB_PLC1_MB_Buffer_DB".Send_CmdSeq := "DB_PLC1_Send_To_PLC2_DB".CmdSeq;
END_REGION

REGION Network 4: Modbus TCP Client - Copy Send Cmd_Start
   RUNG wire#powerrail
      Contact( "DB_PLC1_Send_To_PLC2_DB".Cmd_Start )
      Coil( "DB_PLC1_MB_Buffer_DB".Send_Cmd_Start )
   END_RUNG
   // the same network as SCL:
   "DB_PLC1_MB_Buffer_DB".Send_Cmd_Start := "DB_PLC1_Send_To_PLC2_DB".Cmd_Start;
END_REGION

REGION Network 5: Modbus TCP Client - Copy Send Cmd_Stop
   RUNG wire#powerrail
      Contact( "DB_PLC1_Send_To_PLC2_DB".Cmd_Stop )
      Coil( "DB_PLC1_MB_Buffer_DB".Send_Cmd_Stop )
   END_RUNG
   // the same network as SCL:
   "DB_PLC1_MB_Buffer_DB".Send_Cmd_Stop := "DB_PLC1_Send_To_PLC2_DB".Cmd_Stop;
END_REGION

REGION Network 6: Modbus TCP Client - Copy Send Cmd_Reset
   RUNG wire#powerrail
      Contact( "DB_PLC1_Send_To_PLC2_DB".Cmd_Reset )
      Coil( "DB_PLC1_MB_Buffer_DB".Send_Cmd_Reset )
   END_RUNG
   // the same network as SCL:
   "DB_PLC1_MB_Buffer_DB".Send_Cmd_Reset := "DB_PLC1_Send_To_PLC2_DB".Cmd_Reset;
END_REGION

REGION Network 7: Modbus TCP Client - Copy Send Cmd_EStop
   RUNG wire#powerrail
      Contact( "DB_PLC1_Send_To_PLC2_DB".Cmd_EStop )
      Coil( "DB_PLC1_MB_Buffer_DB".Send_Cmd_EStop )
   END_RUNG
   // the same network as SCL:
   "DB_PLC1_MB_Buffer_DB".Send_Cmd_EStop := "DB_PLC1_Send_To_PLC2_DB".Cmd_EStop;
END_REGION

REGION Network 8: Modbus TCP Client - Copy Send Cmd_Pump_Branch2_To_SubTanks
   RUNG wire#powerrail
      Contact( "DB_PLC1_Send_To_PLC2_DB".Cmd_Pump_Branch2_To_SubTanks )
      Coil( "DB_PLC1_MB_Buffer_DB".Send_Cmd_Pump_Branch2_To_SubTanks )
   END_RUNG
   // the same network as SCL:
   "DB_PLC1_MB_Buffer_DB".Send_Cmd_Pump_Branch2_To_SubTanks := "DB_PLC1_Send_To_PLC2_DB".Cmd_Pump_Branch2_To_SubTanks;
END_REGION

REGION Network 9: Modbus TCP Client - Copy Send Cmd_Load_Recipe
   RUNG wire#powerrail
      Contact( "DB_PLC1_Send_To_PLC2_DB".Cmd_Load_Recipe )
      Coil( "DB_PLC1_MB_Buffer_DB".Send_Cmd_Load_Recipe )
   END_RUNG
   // the same network as SCL:
   "DB_PLC1_MB_Buffer_DB".Send_Cmd_Load_Recipe := "DB_PLC1_Send_To_PLC2_DB".Cmd_Load_Recipe;
END_REGION

REGION Network 10: Modbus TCP Client - Copy Send Heartbeat
   RUNG wire#powerrail
      { S7_GenerateENO := "TRUE" } Move(in := "DB_PLC1_Send_To_PLC2_DB".Heartbeat, out1 => "DB_PLC1_MB_Buffer_DB".Send_Heartbeat)
   END_RUNG
   // the same network as SCL:
   "DB_PLC1_MB_Buffer_DB".Send_Heartbeat := "DB_PLC1_Send_To_PLC2_DB".Heartbeat;
END_REGION

REGION Network 11: PLC1 - Gọi logic khởi tạo recipe mặc định PLC1
   RUNG wire#powerrail
      "FC_Init_Default_Recipe_PLC1"()
   END_RUNG
   // the same network as SCL:
   "FC_Init_Default_Recipe_PLC1"();
END_REGION

REGION Network 12: PLC1 - gọi logic Bồn 1 và Bồn 2
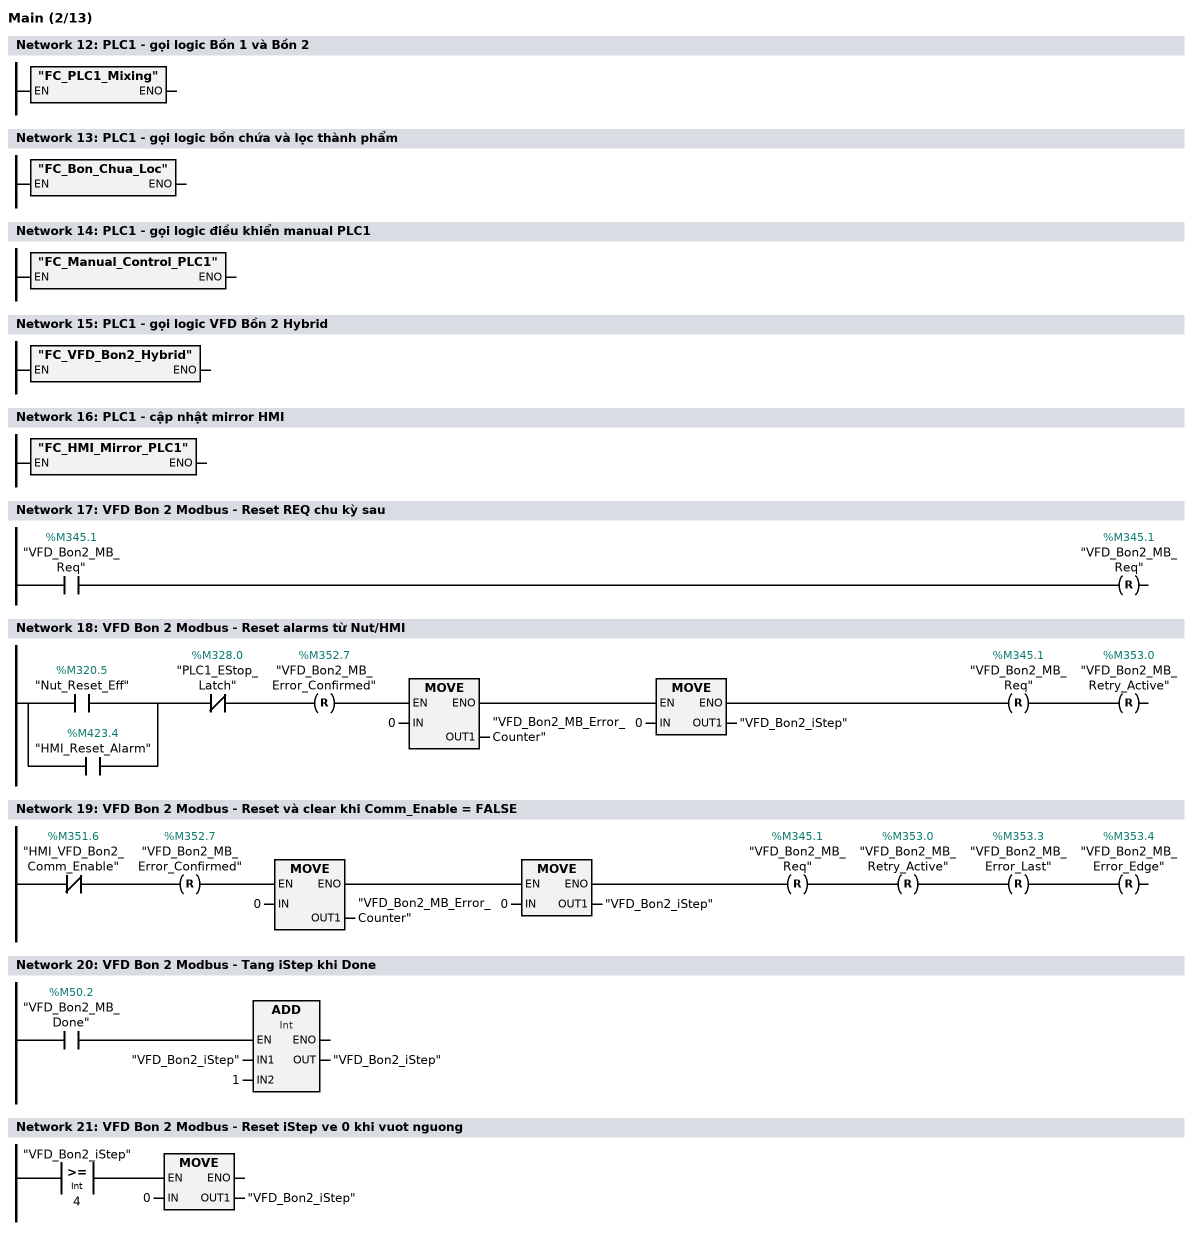
   RUNG wire#powerrail
      "FC_PLC1_Mixing"()
   END_RUNG
   // the same network as SCL:
   "FC_PLC1_Mixing"();
END_REGION

REGION Network 13: PLC1 - gọi logic bồn chứa và lọc thành phẩm
   RUNG wire#powerrail
      "FC_Bon_Chua_Loc"()
   END_RUNG
   // the same network as SCL:
   "FC_Bon_Chua_Loc"();
END_REGION

REGION Network 14: PLC1 - gọi logic điều khiển manual PLC1
   RUNG wire#powerrail
      "FC_Manual_Control_PLC1"()
   END_RUNG
   // the same network as SCL:
   "FC_Manual_Control_PLC1"();
END_REGION

REGION Network 15: PLC1 - gọi logic VFD Bồn 2 Hybrid
   RUNG wire#powerrail
      "FC_VFD_Bon2_Hybrid"()
   END_RUNG
   // the same network as SCL:
   "FC_VFD_Bon2_Hybrid"();
END_REGION

REGION Network 16: PLC1 - cập nhật mirror HMI
   RUNG wire#powerrail
      "FC_HMI_Mirror_PLC1"()
   END_RUNG
   // the same network as SCL:
   "FC_HMI_Mirror_PLC1"();
END_REGION

REGION Network 17: VFD Bon 2 Modbus - Reset REQ chu kỳ sau
   RUNG wire#powerrail
      Contact( "VFD_Bon2_MB_Req" )
      R_Coil( "VFD_Bon2_MB_Req" )
   END_RUNG
   // the same network as SCL:
   IF "VFD_Bon2_MB_Req" THEN "VFD_Bon2_MB_Req" := FALSE; END_IF;
END_REGION

REGION Network 18: VFD Bon 2 Modbus - Reset alarms từ Nut/HMI
   RUNG wire#powerrail
      Contact( "Nut_Reset_Eff" )
      wire#w1
      I_Contact( "PLC1_EStop_Latch" )
      R_Coil( "VFD_Bon2_MB_Error_Confirmed" )
      { S7_GenerateENO := "TRUE" } Move(in := 0, out1 => "VFD_Bon2_MB_Error_Counter")
      { S7_GenerateENO := "TRUE" } Move(in := 0, out1 => "VFD_Bon2_iStep")
      R_Coil( "VFD_Bon2_MB_Req" )
      R_Coil( "VFD_Bon2_MB_Retry_Active" )
   END_RUNG
   RUNG wire#powerrail
      Contact( "HMI_Reset_Alarm" )
   END_RUNG wire#w1
   // the same network as SCL:
   // ENO of a box is taken as its EN; it also drops when the box reports an error
   IF ("Nut_Reset_Eff" OR "HMI_Reset_Alarm") AND NOT "PLC1_EStop_Latch" THEN
       "VFD_Bon2_MB_Error_Confirmed" := FALSE;
       "VFD_Bon2_MB_Error_Counter" := 0;
       "VFD_Bon2_iStep" := 0;
       "VFD_Bon2_MB_Req" := FALSE;
       "VFD_Bon2_MB_Retry_Active" := FALSE;
   END_IF;
END_REGION

REGION Network 19: VFD Bon 2 Modbus - Reset và clear khi Comm_Enable = FALSE
   RUNG wire#powerrail
      I_Contact( "HMI_VFD_Bon2_Comm_Enable" )
      R_Coil( "VFD_Bon2_MB_Error_Confirmed" )
      { S7_GenerateENO := "TRUE" } Move(in := 0, out1 => "VFD_Bon2_MB_Error_Counter")
      { S7_GenerateENO := "TRUE" } Move(in := 0, out1 => "VFD_Bon2_iStep")
      R_Coil( "VFD_Bon2_MB_Req" )
      R_Coil( "VFD_Bon2_MB_Retry_Active" )
      R_Coil( "VFD_Bon2_MB_Error_Last" )
      R_Coil( "VFD_Bon2_MB_Error_Edge" )
   END_RUNG
   // the same network as SCL:
   // ENO of a box is taken as its EN; it also drops when the box reports an error
   IF NOT "HMI_VFD_Bon2_Comm_Enable" THEN
       "VFD_Bon2_MB_Error_Confirmed" := FALSE;
       "VFD_Bon2_MB_Error_Counter" := 0;
       "VFD_Bon2_iStep" := 0;
       "VFD_Bon2_MB_Req" := FALSE;
       "VFD_Bon2_MB_Retry_Active" := FALSE;
       "VFD_Bon2_MB_Error_Last" := FALSE;
       "VFD_Bon2_MB_Error_Edge" := FALSE;
   END_IF;
END_REGION

REGION Network 20: VFD Bon 2 Modbus - Tang iStep khi Done
   RUNG wire#powerrail
      Contact( "VFD_Bon2_MB_Done" )
      { S7_Templates := "SrcType := Int"; S7_GenerateENO := "TRUE" } Add(in1 := "VFD_Bon2_iStep", in2 := 1, out => "VFD_Bon2_iStep")
   END_RUNG
   // the same network as SCL:
   IF "VFD_Bon2_MB_Done" THEN "VFD_Bon2_iStep" := "VFD_Bon2_iStep" + 1; END_IF;
END_REGION

REGION Network 21: VFD Bon 2 Modbus - Reset iStep ve 0 khi vuot nguong
   RUNG wire#powerrail
      { S7_Templates := "SrcType := Int" } GE_Contact(in1 := "VFD_Bon2_iStep", in2 := 4)
      { S7_GenerateENO := "TRUE" } Move(in := 0, out1 => "VFD_Bon2_iStep")
   END_RUNG
   // the same network as SCL:
   IF "VFD_Bon2_iStep" >= 4 THEN "VFD_Bon2_iStep" := 0; END_IF;
END_REGION

REGION Network 22: VFD Bon 2 Modbus - Set REQ khi co trigger
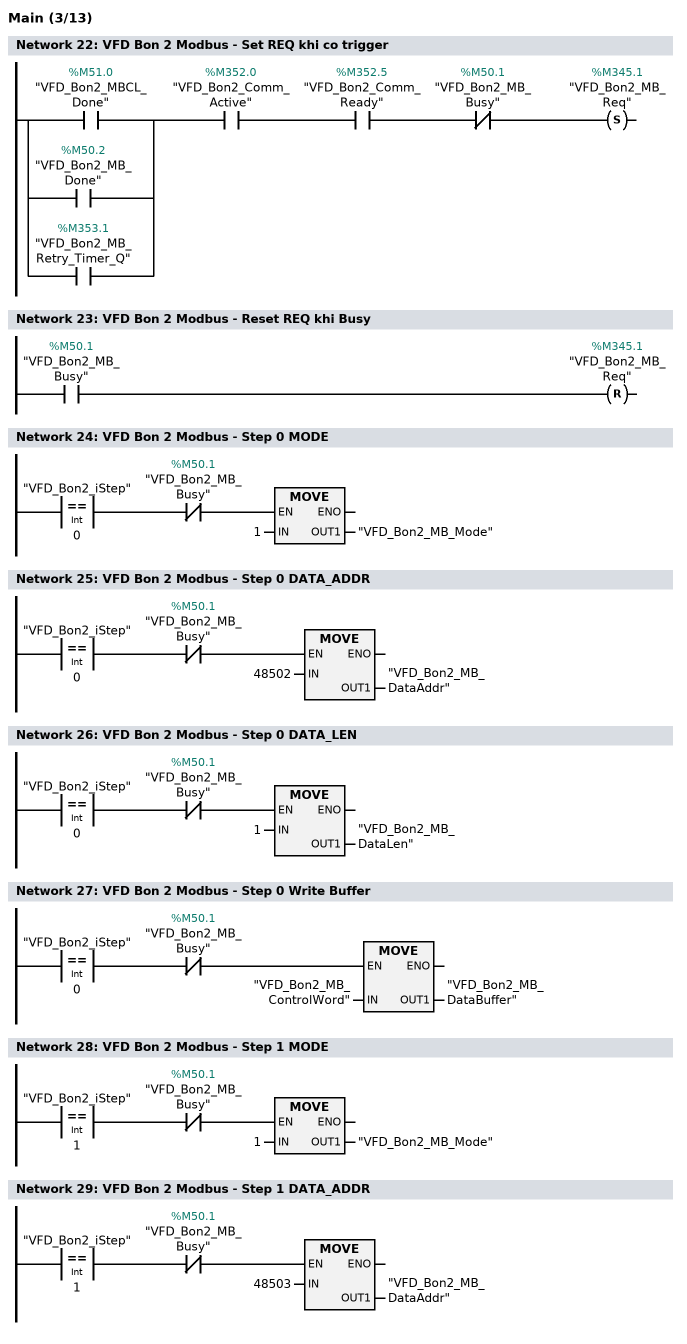
   RUNG wire#powerrail
      Contact( "VFD_Bon2_MBCL_Done" )
      wire#w1
      Contact( "VFD_Bon2_Comm_Active" )
      Contact( "VFD_Bon2_Comm_Ready" )
      I_Contact( "VFD_Bon2_MB_Busy" )
      S_Coil( "VFD_Bon2_MB_Req" )
   END_RUNG
   RUNG wire#powerrail
      Contact( "VFD_Bon2_MB_Done" )
   END_RUNG wire#w1
   RUNG wire#powerrail
      Contact( "VFD_Bon2_MB_Retry_Timer_Q" )
   END_RUNG wire#w1
   // the same network as SCL:
   IF ("VFD_Bon2_MBCL_Done" OR "VFD_Bon2_MB_Done" OR "VFD_Bon2_MB_Retry_Timer_Q") AND "VFD_Bon2_Comm_Active" AND "VFD_Bon2_Comm_Ready" AND NOT "VFD_Bon2_MB_Busy" THEN
       "VFD_Bon2_MB_Req" := TRUE;
   END_IF;
END_REGION

REGION Network 23: VFD Bon 2 Modbus - Reset REQ khi Busy
   RUNG wire#powerrail
      Contact( "VFD_Bon2_MB_Busy" )
      R_Coil( "VFD_Bon2_MB_Req" )
   END_RUNG
   // the same network as SCL:
   IF "VFD_Bon2_MB_Busy" THEN "VFD_Bon2_MB_Req" := FALSE; END_IF;
END_REGION

REGION Network 24: VFD Bon 2 Modbus - Step 0 MODE
   RUNG wire#powerrail
      { S7_Templates := "SrcType := Int" } EQ_Contact(in1 := "VFD_Bon2_iStep", in2 := 0)
      I_Contact( "VFD_Bon2_MB_Busy" )
      { S7_GenerateENO := "TRUE" } Move(in := 1, out1 => "VFD_Bon2_MB_Mode")
   END_RUNG
   // the same network as SCL:
   IF ("VFD_Bon2_iStep" = 0) AND NOT "VFD_Bon2_MB_Busy" THEN "VFD_Bon2_MB_Mode" := 1; END_IF;
END_REGION

REGION Network 25: VFD Bon 2 Modbus - Step 0 DATA_ADDR
   RUNG wire#powerrail
      { S7_Templates := "SrcType := Int" } EQ_Contact(in1 := "VFD_Bon2_iStep", in2 := 0)
      I_Contact( "VFD_Bon2_MB_Busy" )
      { S7_GenerateENO := "TRUE" } Move(in := 48502, out1 => "VFD_Bon2_MB_DataAddr")
   END_RUNG
   // the same network as SCL:
   IF ("VFD_Bon2_iStep" = 0) AND NOT "VFD_Bon2_MB_Busy" THEN "VFD_Bon2_MB_DataAddr" := 48502; END_IF;
END_REGION

REGION Network 26: VFD Bon 2 Modbus - Step 0 DATA_LEN
   RUNG wire#powerrail
      { S7_Templates := "SrcType := Int" } EQ_Contact(in1 := "VFD_Bon2_iStep", in2 := 0)
      I_Contact( "VFD_Bon2_MB_Busy" )
      { S7_GenerateENO := "TRUE" } Move(in := 1, out1 => "VFD_Bon2_MB_DataLen")
   END_RUNG
   // the same network as SCL:
   IF ("VFD_Bon2_iStep" = 0) AND NOT "VFD_Bon2_MB_Busy" THEN "VFD_Bon2_MB_DataLen" := 1; END_IF;
END_REGION

REGION Network 27: VFD Bon 2 Modbus - Step 0 Write Buffer
   RUNG wire#powerrail
      { S7_Templates := "SrcType := Int" } EQ_Contact(in1 := "VFD_Bon2_iStep", in2 := 0)
      I_Contact( "VFD_Bon2_MB_Busy" )
      { S7_GenerateENO := "TRUE" } Move(in := "VFD_Bon2_MB_ControlWord", out1 => "VFD_Bon2_MB_DataBuffer")
   END_RUNG
   // the same network as SCL:
   IF ("VFD_Bon2_iStep" = 0) AND NOT "VFD_Bon2_MB_Busy" THEN
       "VFD_Bon2_MB_DataBuffer" := "VFD_Bon2_MB_ControlWord";
   END_IF;
END_REGION

REGION Network 28: VFD Bon 2 Modbus - Step 1 MODE
   RUNG wire#powerrail
      { S7_Templates := "SrcType := Int" } EQ_Contact(in1 := "VFD_Bon2_iStep", in2 := 1)
      I_Contact( "VFD_Bon2_MB_Busy" )
      { S7_GenerateENO := "TRUE" } Move(in := 1, out1 => "VFD_Bon2_MB_Mode")
   END_RUNG
   // the same network as SCL:
   IF ("VFD_Bon2_iStep" = 1) AND NOT "VFD_Bon2_MB_Busy" THEN "VFD_Bon2_MB_Mode" := 1; END_IF;
END_REGION

REGION Network 29: VFD Bon 2 Modbus - Step 1 DATA_ADDR
   RUNG wire#powerrail
      { S7_Templates := "SrcType := Int" } EQ_Contact(in1 := "VFD_Bon2_iStep", in2 := 1)
      I_Contact( "VFD_Bon2_MB_Busy" )
      { S7_GenerateENO := "TRUE" } Move(in := 48503, out1 => "VFD_Bon2_MB_DataAddr")
   END_RUNG
   // the same network as SCL:
   IF ("VFD_Bon2_iStep" = 1) AND NOT "VFD_Bon2_MB_Busy" THEN "VFD_Bon2_MB_DataAddr" := 48503; END_IF;
END_REGION

REGION Network 30: VFD Bon 2 Modbus - Step 1 DATA_LEN
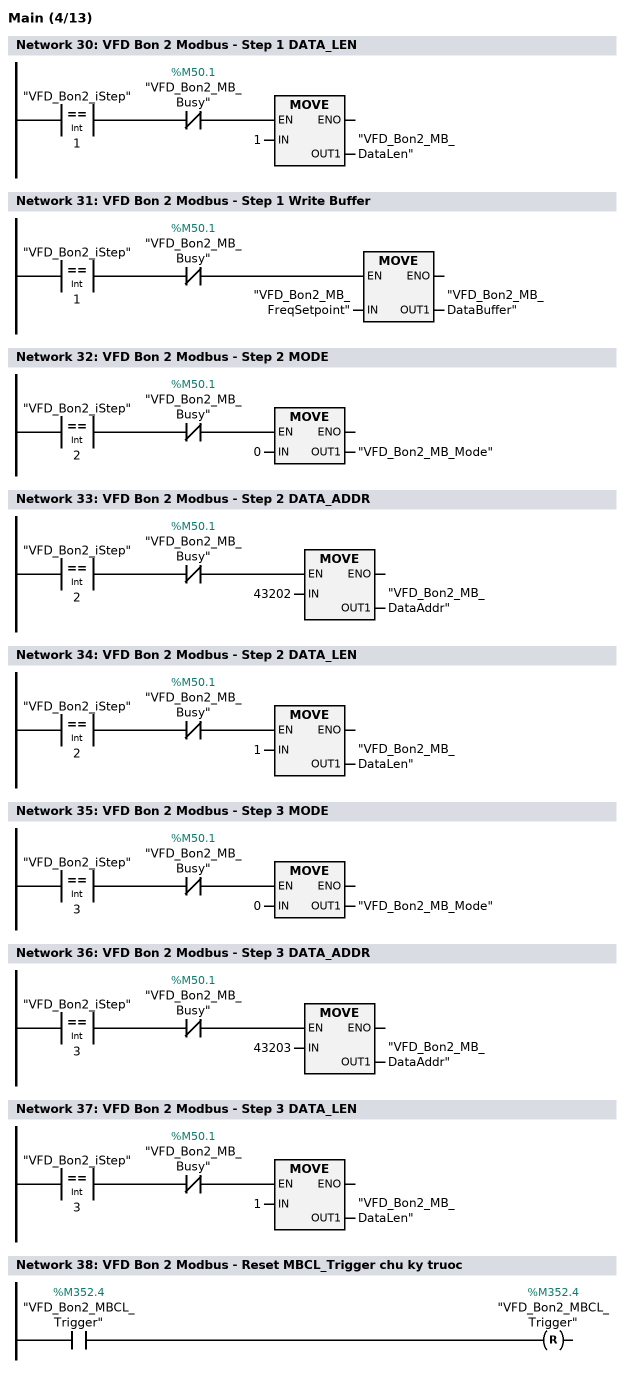
   RUNG wire#powerrail
      { S7_Templates := "SrcType := Int" } EQ_Contact(in1 := "VFD_Bon2_iStep", in2 := 1)
      I_Contact( "VFD_Bon2_MB_Busy" )
      { S7_GenerateENO := "TRUE" } Move(in := 1, out1 => "VFD_Bon2_MB_DataLen")
   END_RUNG
   // the same network as SCL:
   IF ("VFD_Bon2_iStep" = 1) AND NOT "VFD_Bon2_MB_Busy" THEN "VFD_Bon2_MB_DataLen" := 1; END_IF;
END_REGION

REGION Network 31: VFD Bon 2 Modbus - Step 1 Write Buffer
   RUNG wire#powerrail
      { S7_Templates := "SrcType := Int" } EQ_Contact(in1 := "VFD_Bon2_iStep", in2 := 1)
      I_Contact( "VFD_Bon2_MB_Busy" )
      { S7_GenerateENO := "TRUE" } Move(in := "VFD_Bon2_MB_FreqSetpoint", out1 => "VFD_Bon2_MB_DataBuffer")
   END_RUNG
   // the same network as SCL:
   IF ("VFD_Bon2_iStep" = 1) AND NOT "VFD_Bon2_MB_Busy" THEN
       "VFD_Bon2_MB_DataBuffer" := "VFD_Bon2_MB_FreqSetpoint";
   END_IF;
END_REGION

REGION Network 32: VFD Bon 2 Modbus - Step 2 MODE
   RUNG wire#powerrail
      { S7_Templates := "SrcType := Int" } EQ_Contact(in1 := "VFD_Bon2_iStep", in2 := 2)
      I_Contact( "VFD_Bon2_MB_Busy" )
      { S7_GenerateENO := "TRUE" } Move(in := 0, out1 => "VFD_Bon2_MB_Mode")
   END_RUNG
   // the same network as SCL:
   IF ("VFD_Bon2_iStep" = 2) AND NOT "VFD_Bon2_MB_Busy" THEN "VFD_Bon2_MB_Mode" := 0; END_IF;
END_REGION

REGION Network 33: VFD Bon 2 Modbus - Step 2 DATA_ADDR
   RUNG wire#powerrail
      { S7_Templates := "SrcType := Int" } EQ_Contact(in1 := "VFD_Bon2_iStep", in2 := 2)
      I_Contact( "VFD_Bon2_MB_Busy" )
      { S7_GenerateENO := "TRUE" } Move(in := 43202, out1 => "VFD_Bon2_MB_DataAddr")
   END_RUNG
   // the same network as SCL:
   IF ("VFD_Bon2_iStep" = 2) AND NOT "VFD_Bon2_MB_Busy" THEN "VFD_Bon2_MB_DataAddr" := 43202; END_IF;
END_REGION

REGION Network 34: VFD Bon 2 Modbus - Step 2 DATA_LEN
   RUNG wire#powerrail
      { S7_Templates := "SrcType := Int" } EQ_Contact(in1 := "VFD_Bon2_iStep", in2 := 2)
      I_Contact( "VFD_Bon2_MB_Busy" )
      { S7_GenerateENO := "TRUE" } Move(in := 1, out1 => "VFD_Bon2_MB_DataLen")
   END_RUNG
   // the same network as SCL:
   IF ("VFD_Bon2_iStep" = 2) AND NOT "VFD_Bon2_MB_Busy" THEN "VFD_Bon2_MB_DataLen" := 1; END_IF;
END_REGION

REGION Network 35: VFD Bon 2 Modbus - Step 3 MODE
   RUNG wire#powerrail
      { S7_Templates := "SrcType := Int" } EQ_Contact(in1 := "VFD_Bon2_iStep", in2 := 3)
      I_Contact( "VFD_Bon2_MB_Busy" )
      { S7_GenerateENO := "TRUE" } Move(in := 0, out1 => "VFD_Bon2_MB_Mode")
   END_RUNG
   // the same network as SCL:
   IF ("VFD_Bon2_iStep" = 3) AND NOT "VFD_Bon2_MB_Busy" THEN "VFD_Bon2_MB_Mode" := 0; END_IF;
END_REGION

REGION Network 36: VFD Bon 2 Modbus - Step 3 DATA_ADDR
   RUNG wire#powerrail
      { S7_Templates := "SrcType := Int" } EQ_Contact(in1 := "VFD_Bon2_iStep", in2 := 3)
      I_Contact( "VFD_Bon2_MB_Busy" )
      { S7_GenerateENO := "TRUE" } Move(in := 43203, out1 => "VFD_Bon2_MB_DataAddr")
   END_RUNG
   // the same network as SCL:
   IF ("VFD_Bon2_iStep" = 3) AND NOT "VFD_Bon2_MB_Busy" THEN "VFD_Bon2_MB_DataAddr" := 43203; END_IF;
END_REGION

REGION Network 37: VFD Bon 2 Modbus - Step 3 DATA_LEN
   RUNG wire#powerrail
      { S7_Templates := "SrcType := Int" } EQ_Contact(in1 := "VFD_Bon2_iStep", in2 := 3)
      I_Contact( "VFD_Bon2_MB_Busy" )
      { S7_GenerateENO := "TRUE" } Move(in := 1, out1 => "VFD_Bon2_MB_DataLen")
   END_RUNG
   // the same network as SCL:
   IF ("VFD_Bon2_iStep" = 3) AND NOT "VFD_Bon2_MB_Busy" THEN "VFD_Bon2_MB_DataLen" := 1; END_IF;
END_REGION

REGION Network 38: VFD Bon 2 Modbus - Reset MBCL_Trigger chu ky truoc
   RUNG wire#powerrail
      Contact( "VFD_Bon2_MBCL_Trigger" )
      R_Coil( "VFD_Bon2_MBCL_Trigger" )
   END_RUNG
   // the same network as SCL:
   IF "VFD_Bon2_MBCL_Trigger" THEN "VFD_Bon2_MBCL_Trigger" := FALSE; END_IF;
END_REGION

REGION Network 39: VFD Bon 2 Modbus - Trigger MB_COMM_LOAD khi delay contactor xong
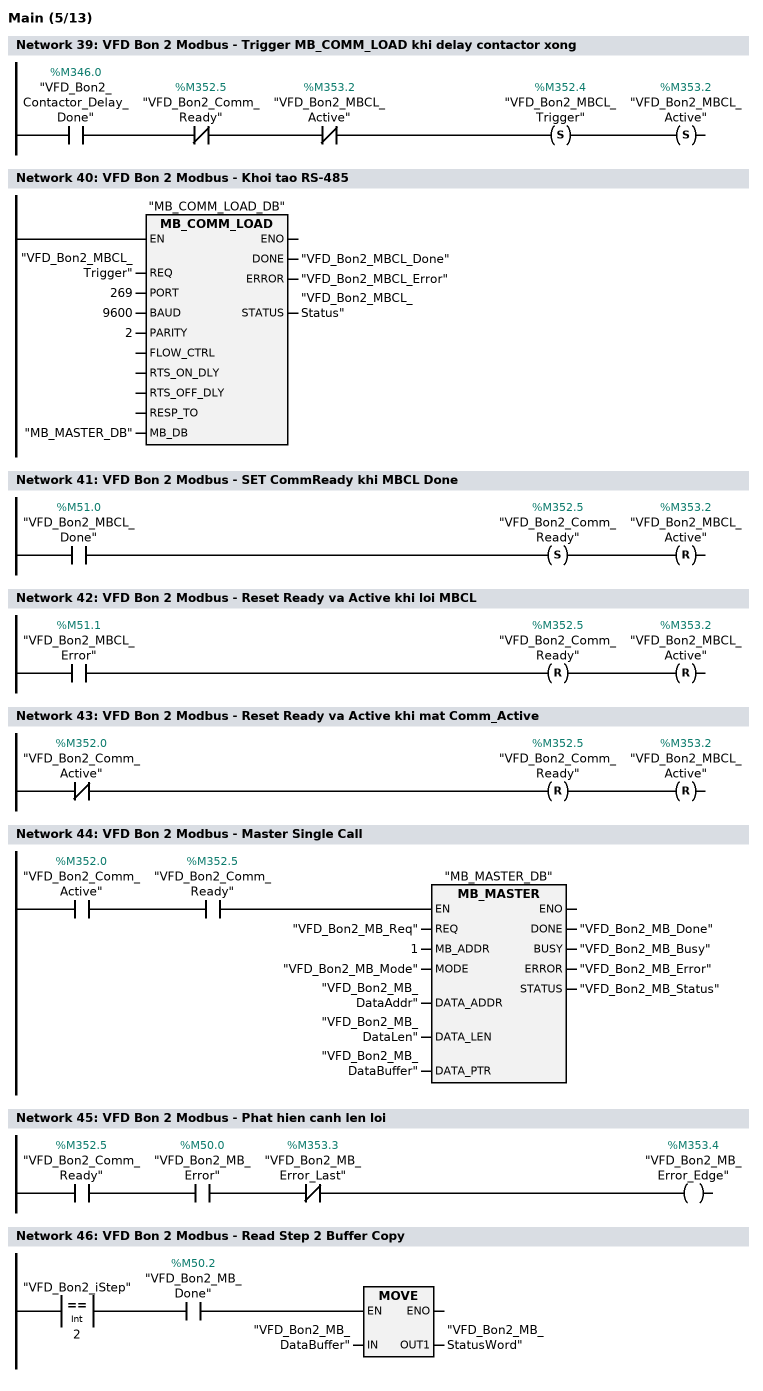
   RUNG wire#powerrail
      Contact( "VFD_Bon2_Contactor_Delay_Done" )
      I_Contact( "VFD_Bon2_Comm_Ready" )
      I_Contact( "VFD_Bon2_MBCL_Active" )
      S_Coil( "VFD_Bon2_MBCL_Trigger" )
      S_Coil( "VFD_Bon2_MBCL_Active" )
   END_RUNG
   // the same network as SCL:
   IF "VFD_Bon2_Contactor_Delay_Done" AND NOT "VFD_Bon2_Comm_Ready" AND NOT "VFD_Bon2_MBCL_Active" THEN
       "VFD_Bon2_MBCL_Trigger" := TRUE;
       "VFD_Bon2_MBCL_Active" := TRUE;
   END_IF;
END_REGION

REGION Network 40: VFD Bon 2 Modbus - Khoi tao RS-485
   RUNG wire#powerrail
      "MB_COMM_LOAD_DB".MB_COMM_LOAD(REQ := "VFD_Bon2_MBCL_Trigger", PORT := 269, BAUD := 9600, PARITY := 2, FLOW_CTRL :=, RTS_ON_DLY :=, RTS_OFF_DLY :=, RESP_TO :=, MB_DB := "MB_MASTER_DB", DONE => "VFD_Bon2_MBCL_Done", ERROR => "VFD_Bon2_MBCL_Error", STATUS => "VFD_Bon2_MBCL_Status")
   END_RUNG
   // the same network as SCL:
   "MB_COMM_LOAD_DB"(REQ := "VFD_Bon2_MBCL_Trigger",   // MB_COMM_LOAD
                     PORT := 269,
                     BAUD := 9600,
                     PARITY := 2,
                     MB_DB := "MB_MASTER_DB",
                     DONE => "VFD_Bon2_MBCL_Done",
                     ERROR => "VFD_Bon2_MBCL_Error",
                     STATUS => "VFD_Bon2_MBCL_Status");
END_REGION

REGION Network 41: VFD Bon 2 Modbus - SET CommReady khi MBCL Done
   RUNG wire#powerrail
      Contact( "VFD_Bon2_MBCL_Done" )
      S_Coil( "VFD_Bon2_Comm_Ready" )
      R_Coil( "VFD_Bon2_MBCL_Active" )
   END_RUNG
   // the same network as SCL:
   IF "VFD_Bon2_MBCL_Done" THEN
       "VFD_Bon2_Comm_Ready" := TRUE;
       "VFD_Bon2_MBCL_Active" := FALSE;
   END_IF;
END_REGION

REGION Network 42: VFD Bon 2 Modbus - Reset Ready va Active khi loi MBCL
   RUNG wire#powerrail
      Contact( "VFD_Bon2_MBCL_Error" )
      R_Coil( "VFD_Bon2_Comm_Ready" )
      R_Coil( "VFD_Bon2_MBCL_Active" )
   END_RUNG
   // the same network as SCL:
   IF "VFD_Bon2_MBCL_Error" THEN
       "VFD_Bon2_Comm_Ready" := FALSE;
       "VFD_Bon2_MBCL_Active" := FALSE;
   END_IF;
END_REGION

REGION Network 43: VFD Bon 2 Modbus - Reset Ready va Active khi mat Comm_Active
   RUNG wire#powerrail
      I_Contact( "VFD_Bon2_Comm_Active" )
      R_Coil( "VFD_Bon2_Comm_Ready" )
      R_Coil( "VFD_Bon2_MBCL_Active" )
   END_RUNG
   // the same network as SCL:
   IF NOT "VFD_Bon2_Comm_Active" THEN
       "VFD_Bon2_Comm_Ready" := FALSE;
       "VFD_Bon2_MBCL_Active" := FALSE;
   END_IF;
END_REGION

REGION Network 44: VFD Bon 2 Modbus - Master Single Call
   RUNG wire#powerrail
      Contact( "VFD_Bon2_Comm_Active" )
      Contact( "VFD_Bon2_Comm_Ready" )
      "MB_MASTER_DB".MB_MASTER(REQ := "VFD_Bon2_MB_Req", MB_ADDR := 1, MODE := "VFD_Bon2_MB_Mode", DATA_ADDR := "VFD_Bon2_MB_DataAddr", DATA_LEN := "VFD_Bon2_MB_DataLen", DATA_PTR := "VFD_Bon2_MB_DataBuffer", DONE => "VFD_Bon2_MB_Done", BUSY => "VFD_Bon2_MB_Busy", ERROR => "VFD_Bon2_MB_Error", STATUS => "VFD_Bon2_MB_Status")
   END_RUNG
   // the same network as SCL:
   IF "VFD_Bon2_Comm_Active" AND "VFD_Bon2_Comm_Ready" THEN
       "MB_MASTER_DB"(REQ := "VFD_Bon2_MB_Req",   // MB_MASTER
                      MB_ADDR := 1,
                      MODE := "VFD_Bon2_MB_Mode",
                      DATA_ADDR := "VFD_Bon2_MB_DataAddr",
                      DATA_LEN := "VFD_Bon2_MB_DataLen",
                      DATA_PTR := "VFD_Bon2_MB_DataBuffer",
                      DONE => "VFD_Bon2_MB_Done",
                      BUSY => "VFD_Bon2_MB_Busy",
                      ERROR => "VFD_Bon2_MB_Error",
                      STATUS => "VFD_Bon2_MB_Status");
   END_IF;
END_REGION

REGION Network 45: VFD Bon 2 Modbus - Phat hien canh len loi
   RUNG wire#powerrail
      Contact( "VFD_Bon2_Comm_Ready" )
      Contact( "VFD_Bon2_MB_Error" )
      I_Contact( "VFD_Bon2_MB_Error_Last" )
      Coil( "VFD_Bon2_MB_Error_Edge" )
   END_RUNG
   // the same network as SCL:
   "VFD_Bon2_MB_Error_Edge" := "VFD_Bon2_Comm_Ready" AND "VFD_Bon2_MB_Error" AND NOT "VFD_Bon2_MB_Error_Last";
END_REGION

REGION Network 46: VFD Bon 2 Modbus - Read Step 2 Buffer Copy
   RUNG wire#powerrail
      { S7_Templates := "SrcType := Int" } EQ_Contact(in1 := "VFD_Bon2_iStep", in2 := 2)
      Contact( "VFD_Bon2_MB_Done" )
      { S7_GenerateENO := "TRUE" } Move(in := "VFD_Bon2_MB_DataBuffer", out1 => "VFD_Bon2_MB_StatusWord")
   END_RUNG
   // the same network as SCL:
   IF ("VFD_Bon2_iStep" = 2) AND "VFD_Bon2_MB_Done" THEN
       "VFD_Bon2_MB_StatusWord" := "VFD_Bon2_MB_DataBuffer";
   END_IF;
END_REGION

REGION Network 47: VFD Bon 2 Modbus - Read Step 3 Buffer Copy
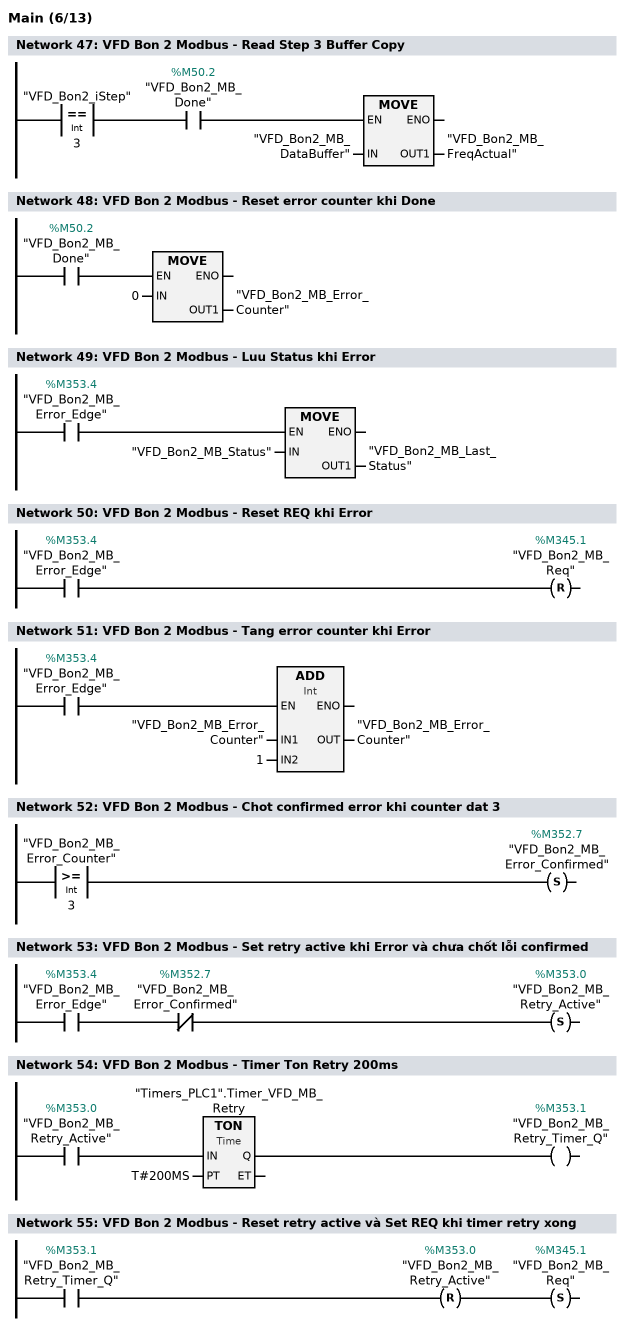
   RUNG wire#powerrail
      { S7_Templates := "SrcType := Int" } EQ_Contact(in1 := "VFD_Bon2_iStep", in2 := 3)
      Contact( "VFD_Bon2_MB_Done" )
      { S7_GenerateENO := "TRUE" } Move(in := "VFD_Bon2_MB_DataBuffer", out1 => "VFD_Bon2_MB_FreqActual")
   END_RUNG
   // the same network as SCL:
   IF ("VFD_Bon2_iStep" = 3) AND "VFD_Bon2_MB_Done" THEN
       "VFD_Bon2_MB_FreqActual" := "VFD_Bon2_MB_DataBuffer";
   END_IF;
END_REGION

REGION Network 48: VFD Bon 2 Modbus - Reset error counter khi Done
   RUNG wire#powerrail
      Contact( "VFD_Bon2_MB_Done" )
      { S7_GenerateENO := "TRUE" } Move(in := 0, out1 => "VFD_Bon2_MB_Error_Counter")
   END_RUNG
   // the same network as SCL:
   IF "VFD_Bon2_MB_Done" THEN "VFD_Bon2_MB_Error_Counter" := 0; END_IF;
END_REGION

REGION Network 49: VFD Bon 2 Modbus - Luu Status khi Error
   RUNG wire#powerrail
      Contact( "VFD_Bon2_MB_Error_Edge" )
      { S7_GenerateENO := "TRUE" } Move(in := "VFD_Bon2_MB_Status", out1 => "VFD_Bon2_MB_Last_Status")
   END_RUNG
   // the same network as SCL:
   IF "VFD_Bon2_MB_Error_Edge" THEN "VFD_Bon2_MB_Last_Status" := "VFD_Bon2_MB_Status"; END_IF;
END_REGION

REGION Network 50: VFD Bon 2 Modbus - Reset REQ khi Error
   RUNG wire#powerrail
      Contact( "VFD_Bon2_MB_Error_Edge" )
      R_Coil( "VFD_Bon2_MB_Req" )
   END_RUNG
   // the same network as SCL:
   IF "VFD_Bon2_MB_Error_Edge" THEN "VFD_Bon2_MB_Req" := FALSE; END_IF;
END_REGION

REGION Network 51: VFD Bon 2 Modbus - Tang error counter khi Error
   RUNG wire#powerrail
      Contact( "VFD_Bon2_MB_Error_Edge" )
      { S7_Templates := "SrcType := Int"; S7_GenerateENO := "TRUE" } Add(in1 := "VFD_Bon2_MB_Error_Counter", in2 := 1, out => "VFD_Bon2_MB_Error_Counter")
   END_RUNG
   // the same network as SCL:
   IF "VFD_Bon2_MB_Error_Edge" THEN "VFD_Bon2_MB_Error_Counter" := "VFD_Bon2_MB_Error_Counter" + 1; END_IF;
END_REGION

REGION Network 52: VFD Bon 2 Modbus - Chot confirmed error khi counter dat 3
   RUNG wire#powerrail
      { S7_Templates := "SrcType := Int" } GE_Contact(in1 := "VFD_Bon2_MB_Error_Counter", in2 := 3)
      S_Coil( "VFD_Bon2_MB_Error_Confirmed" )
   END_RUNG
   // the same network as SCL:
   IF "VFD_Bon2_MB_Error_Counter" >= 3 THEN "VFD_Bon2_MB_Error_Confirmed" := TRUE; END_IF;
END_REGION

REGION Network 53: VFD Bon 2 Modbus - Set retry active khi Error và chưa chốt lỗi confirmed
   RUNG wire#powerrail
      Contact( "VFD_Bon2_MB_Error_Edge" )
      I_Contact( "VFD_Bon2_MB_Error_Confirmed" )
      S_Coil( "VFD_Bon2_MB_Retry_Active" )
   END_RUNG
   // the same network as SCL:
   IF "VFD_Bon2_MB_Error_Edge" AND NOT "VFD_Bon2_MB_Error_Confirmed" THEN
       "VFD_Bon2_MB_Retry_Active" := TRUE;
   END_IF;
END_REGION

REGION Network 54: VFD Bon 2 Modbus - Timer Ton Retry 200ms
   RUNG wire#powerrail
      Contact( "VFD_Bon2_MB_Retry_Active" )
      { S7_Templates := "time_type := Time" } "Timers_PLC1".Timer_VFD_MB_Retry.TON(pt := T#200MS, et =>)
      Coil( "VFD_Bon2_MB_Retry_Timer_Q" )
   END_RUNG
   // the same network as SCL:
   "Timers_PLC1".Timer_VFD_MB_Retry.TON(IN := "VFD_Bon2_MB_Retry_Active", PT := T#200MS);
   "VFD_Bon2_MB_Retry_Timer_Q" := "Timers_PLC1".Timer_VFD_MB_Retry.Q;
END_REGION

REGION Network 55: VFD Bon 2 Modbus - Reset retry active và Set REQ khi timer retry xong
   RUNG wire#powerrail
      Contact( "VFD_Bon2_MB_Retry_Timer_Q" )
      R_Coil( "VFD_Bon2_MB_Retry_Active" )
      S_Coil( "VFD_Bon2_MB_Req" )
   END_RUNG
   // the same network as SCL:
   IF "VFD_Bon2_MB_Retry_Timer_Q" THEN
       "VFD_Bon2_MB_Retry_Active" := FALSE;
       "VFD_Bon2_MB_Req" := TRUE;
   END_IF;
END_REGION

REGION Network 56: VFD Bon 2 Modbus - Save Error Last State
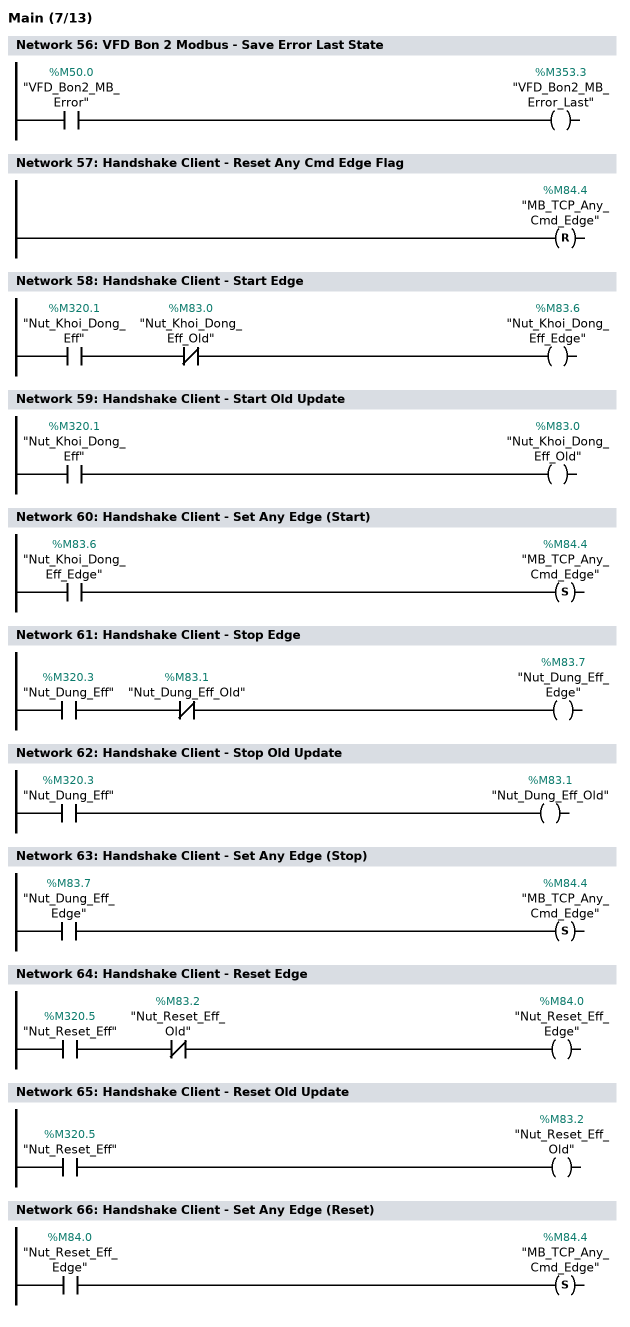
   RUNG wire#powerrail
      Contact( "VFD_Bon2_MB_Error" )
      Coil( "VFD_Bon2_MB_Error_Last" )
   END_RUNG
   // the same network as SCL:
   "VFD_Bon2_MB_Error_Last" := "VFD_Bon2_MB_Error";
END_REGION

REGION Network 57: Handshake Client - Reset Any Cmd Edge Flag
   RUNG wire#powerrail
      R_Coil( "MB_TCP_Any_Cmd_Edge" )
   END_RUNG
   // the same network as SCL:
   "MB_TCP_Any_Cmd_Edge" := FALSE;
END_REGION

REGION Network 58: Handshake Client - Start Edge
   RUNG wire#powerrail
      Contact( "Nut_Khoi_Dong_Eff" )
      I_Contact( "Nut_Khoi_Dong_Eff_Old" )
      Coil( "Nut_Khoi_Dong_Eff_Edge" )
   END_RUNG
   // the same network as SCL:
   "Nut_Khoi_Dong_Eff_Edge" := "Nut_Khoi_Dong_Eff" AND NOT "Nut_Khoi_Dong_Eff_Old";
END_REGION

REGION Network 59: Handshake Client - Start Old Update
   RUNG wire#powerrail
      Contact( "Nut_Khoi_Dong_Eff" )
      Coil( "Nut_Khoi_Dong_Eff_Old" )
   END_RUNG
   // the same network as SCL:
   "Nut_Khoi_Dong_Eff_Old" := "Nut_Khoi_Dong_Eff";
END_REGION

REGION Network 60: Handshake Client - Set Any Edge (Start)
   RUNG wire#powerrail
      Contact( "Nut_Khoi_Dong_Eff_Edge" )
      S_Coil( "MB_TCP_Any_Cmd_Edge" )
   END_RUNG
   // the same network as SCL:
   IF "Nut_Khoi_Dong_Eff_Edge" THEN "MB_TCP_Any_Cmd_Edge" := TRUE; END_IF;
END_REGION

REGION Network 61: Handshake Client - Stop Edge
   RUNG wire#powerrail
      Contact( "Nut_Dung_Eff" )
      I_Contact( "Nut_Dung_Eff_Old" )
      Coil( "Nut_Dung_Eff_Edge" )
   END_RUNG
   // the same network as SCL:
   "Nut_Dung_Eff_Edge" := "Nut_Dung_Eff" AND NOT "Nut_Dung_Eff_Old";
END_REGION

REGION Network 62: Handshake Client - Stop Old Update
   RUNG wire#powerrail
      Contact( "Nut_Dung_Eff" )
      Coil( "Nut_Dung_Eff_Old" )
   END_RUNG
   // the same network as SCL:
   "Nut_Dung_Eff_Old" := "Nut_Dung_Eff";
END_REGION

REGION Network 63: Handshake Client - Set Any Edge (Stop)
   RUNG wire#powerrail
      Contact( "Nut_Dung_Eff_Edge" )
      S_Coil( "MB_TCP_Any_Cmd_Edge" )
   END_RUNG
   // the same network as SCL:
   IF "Nut_Dung_Eff_Edge" THEN "MB_TCP_Any_Cmd_Edge" := TRUE; END_IF;
END_REGION

REGION Network 64: Handshake Client - Reset Edge
   RUNG wire#powerrail
      Contact( "Nut_Reset_Eff" )
      I_Contact( "Nut_Reset_Eff_Old" )
      Coil( "Nut_Reset_Eff_Edge" )
   END_RUNG
   // the same network as SCL:
   "Nut_Reset_Eff_Edge" := "Nut_Reset_Eff" AND NOT "Nut_Reset_Eff_Old";
END_REGION

REGION Network 65: Handshake Client - Reset Old Update
   RUNG wire#powerrail
      Contact( "Nut_Reset_Eff" )
      Coil( "Nut_Reset_Eff_Old" )
   END_RUNG
   // the same network as SCL:
   "Nut_Reset_Eff_Old" := "Nut_Reset_Eff";
END_REGION

REGION Network 66: Handshake Client - Set Any Edge (Reset)
   RUNG wire#powerrail
      Contact( "Nut_Reset_Eff_Edge" )
      S_Coil( "MB_TCP_Any_Cmd_Edge" )
   END_RUNG
   // the same network as SCL:
   IF "Nut_Reset_Eff_Edge" THEN "MB_TCP_Any_Cmd_Edge" := TRUE; END_IF;
END_REGION

REGION Network 67: Handshake Client - EStop Edge
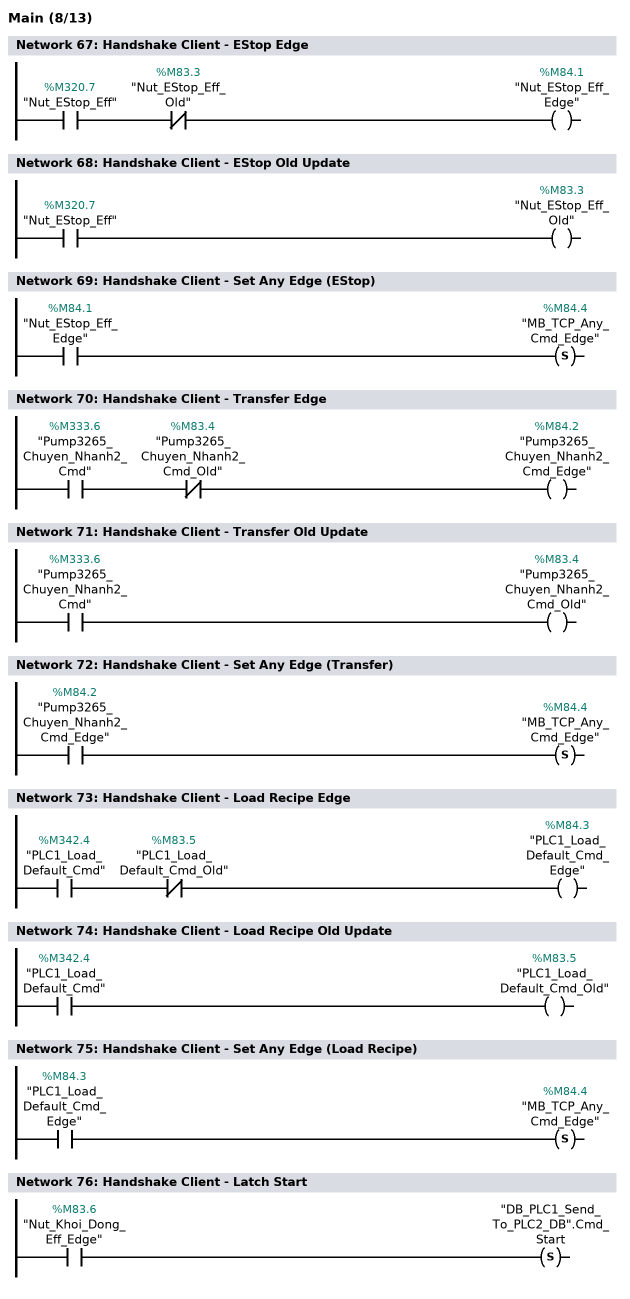
   RUNG wire#powerrail
      Contact( "Nut_EStop_Eff" )
      I_Contact( "Nut_EStop_Eff_Old" )
      Coil( "Nut_EStop_Eff_Edge" )
   END_RUNG
   // the same network as SCL:
   "Nut_EStop_Eff_Edge" := "Nut_EStop_Eff" AND NOT "Nut_EStop_Eff_Old";
END_REGION

REGION Network 68: Handshake Client - EStop Old Update
   RUNG wire#powerrail
      Contact( "Nut_EStop_Eff" )
      Coil( "Nut_EStop_Eff_Old" )
   END_RUNG
   // the same network as SCL:
   "Nut_EStop_Eff_Old" := "Nut_EStop_Eff";
END_REGION

REGION Network 69: Handshake Client - Set Any Edge (EStop)
   RUNG wire#powerrail
      Contact( "Nut_EStop_Eff_Edge" )
      S_Coil( "MB_TCP_Any_Cmd_Edge" )
   END_RUNG
   // the same network as SCL:
   IF "Nut_EStop_Eff_Edge" THEN "MB_TCP_Any_Cmd_Edge" := TRUE; END_IF;
END_REGION

REGION Network 70: Handshake Client - Transfer Edge
   RUNG wire#powerrail
      Contact( "Pump3265_Chuyen_Nhanh2_Cmd" )
      I_Contact( "Pump3265_Chuyen_Nhanh2_Cmd_Old" )
      Coil( "Pump3265_Chuyen_Nhanh2_Cmd_Edge" )
   END_RUNG
   // the same network as SCL:
   "Pump3265_Chuyen_Nhanh2_Cmd_Edge" := "Pump3265_Chuyen_Nhanh2_Cmd" AND NOT "Pump3265_Chuyen_Nhanh2_Cmd_Old";
END_REGION

REGION Network 71: Handshake Client - Transfer Old Update
   RUNG wire#powerrail
      Contact( "Pump3265_Chuyen_Nhanh2_Cmd" )
      Coil( "Pump3265_Chuyen_Nhanh2_Cmd_Old" )
   END_RUNG
   // the same network as SCL:
   "Pump3265_Chuyen_Nhanh2_Cmd_Old" := "Pump3265_Chuyen_Nhanh2_Cmd";
END_REGION

REGION Network 72: Handshake Client - Set Any Edge (Transfer)
   RUNG wire#powerrail
      Contact( "Pump3265_Chuyen_Nhanh2_Cmd_Edge" )
      S_Coil( "MB_TCP_Any_Cmd_Edge" )
   END_RUNG
   // the same network as SCL:
   IF "Pump3265_Chuyen_Nhanh2_Cmd_Edge" THEN "MB_TCP_Any_Cmd_Edge" := TRUE; END_IF;
END_REGION

REGION Network 73: Handshake Client - Load Recipe Edge
   RUNG wire#powerrail
      Contact( "PLC1_Load_Default_Cmd" )
      I_Contact( "PLC1_Load_Default_Cmd_Old" )
      Coil( "PLC1_Load_Default_Cmd_Edge" )
   END_RUNG
   // the same network as SCL:
   "PLC1_Load_Default_Cmd_Edge" := "PLC1_Load_Default_Cmd" AND NOT "PLC1_Load_Default_Cmd_Old";
END_REGION

REGION Network 74: Handshake Client - Load Recipe Old Update
   RUNG wire#powerrail
      Contact( "PLC1_Load_Default_Cmd" )
      Coil( "PLC1_Load_Default_Cmd_Old" )
   END_RUNG
   // the same network as SCL:
   "PLC1_Load_Default_Cmd_Old" := "PLC1_Load_Default_Cmd";
END_REGION

REGION Network 75: Handshake Client - Set Any Edge (Load Recipe)
   RUNG wire#powerrail
      Contact( "PLC1_Load_Default_Cmd_Edge" )
      S_Coil( "MB_TCP_Any_Cmd_Edge" )
   END_RUNG
   // the same network as SCL:
   IF "PLC1_Load_Default_Cmd_Edge" THEN "MB_TCP_Any_Cmd_Edge" := TRUE; END_IF;
END_REGION

REGION Network 76: Handshake Client - Latch Start
   RUNG wire#powerrail
      Contact( "Nut_Khoi_Dong_Eff_Edge" )
      S_Coil( "DB_PLC1_Send_To_PLC2_DB".Cmd_Start )
   END_RUNG
   // the same network as SCL:
   IF "Nut_Khoi_Dong_Eff_Edge" THEN "DB_PLC1_Send_To_PLC2_DB".Cmd_Start := TRUE; END_IF;
END_REGION

REGION Network 77: Handshake Client - Latch Stop
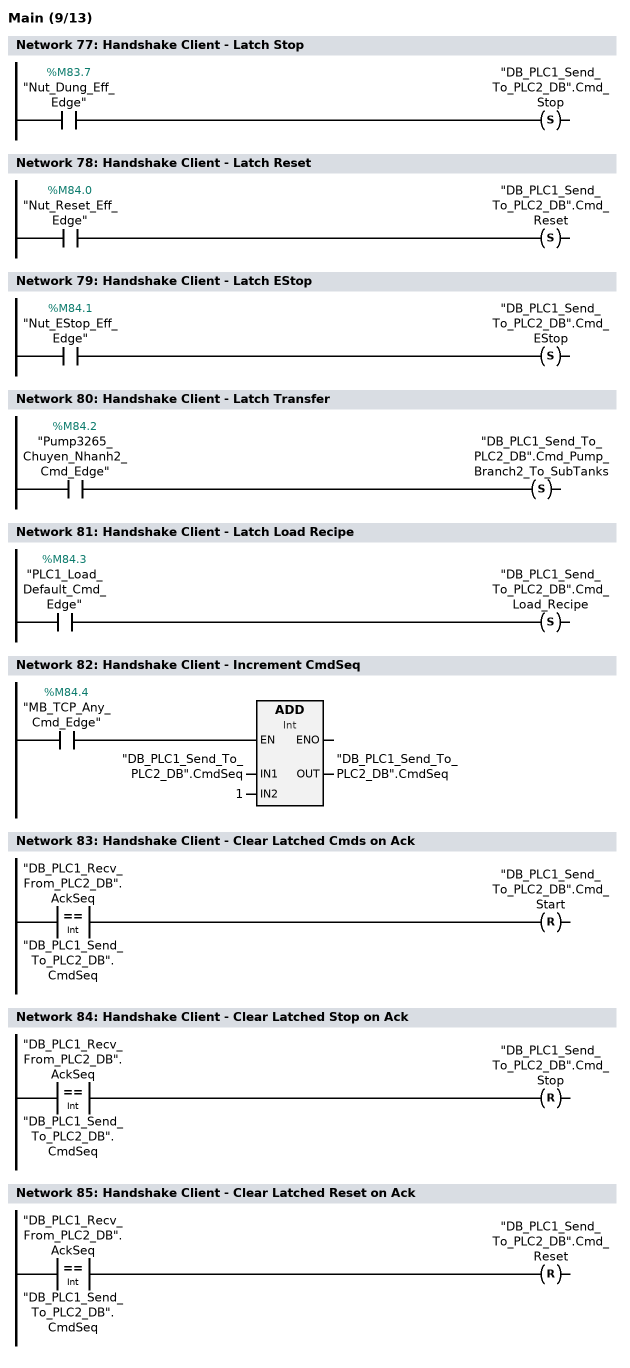
   RUNG wire#powerrail
      Contact( "Nut_Dung_Eff_Edge" )
      S_Coil( "DB_PLC1_Send_To_PLC2_DB".Cmd_Stop )
   END_RUNG
   // the same network as SCL:
   IF "Nut_Dung_Eff_Edge" THEN "DB_PLC1_Send_To_PLC2_DB".Cmd_Stop := TRUE; END_IF;
END_REGION

REGION Network 78: Handshake Client - Latch Reset
   RUNG wire#powerrail
      Contact( "Nut_Reset_Eff_Edge" )
      S_Coil( "DB_PLC1_Send_To_PLC2_DB".Cmd_Reset )
   END_RUNG
   // the same network as SCL:
   IF "Nut_Reset_Eff_Edge" THEN "DB_PLC1_Send_To_PLC2_DB".Cmd_Reset := TRUE; END_IF;
END_REGION

REGION Network 79: Handshake Client - Latch EStop
   RUNG wire#powerrail
      Contact( "Nut_EStop_Eff_Edge" )
      S_Coil( "DB_PLC1_Send_To_PLC2_DB".Cmd_EStop )
   END_RUNG
   // the same network as SCL:
   IF "Nut_EStop_Eff_Edge" THEN "DB_PLC1_Send_To_PLC2_DB".Cmd_EStop := TRUE; END_IF;
END_REGION

REGION Network 80: Handshake Client - Latch Transfer
   RUNG wire#powerrail
      Contact( "Pump3265_Chuyen_Nhanh2_Cmd_Edge" )
      S_Coil( "DB_PLC1_Send_To_PLC2_DB".Cmd_Pump_Branch2_To_SubTanks )
   END_RUNG
   // the same network as SCL:
   IF "Pump3265_Chuyen_Nhanh2_Cmd_Edge" THEN
       "DB_PLC1_Send_To_PLC2_DB".Cmd_Pump_Branch2_To_SubTanks := TRUE;
   END_IF;
END_REGION

REGION Network 81: Handshake Client - Latch Load Recipe
   RUNG wire#powerrail
      Contact( "PLC1_Load_Default_Cmd_Edge" )
      S_Coil( "DB_PLC1_Send_To_PLC2_DB".Cmd_Load_Recipe )
   END_RUNG
   // the same network as SCL:
   IF "PLC1_Load_Default_Cmd_Edge" THEN "DB_PLC1_Send_To_PLC2_DB".Cmd_Load_Recipe := TRUE; END_IF;
END_REGION

REGION Network 82: Handshake Client - Increment CmdSeq
   RUNG wire#powerrail
      Contact( "MB_TCP_Any_Cmd_Edge" )
      { S7_Templates := "SrcType := Int"; S7_GenerateENO := "TRUE" } Add(in1 := "DB_PLC1_Send_To_PLC2_DB".CmdSeq, in2 := 1, out => "DB_PLC1_Send_To_PLC2_DB".CmdSeq)
   END_RUNG
   // the same network as SCL:
   IF "MB_TCP_Any_Cmd_Edge" THEN
       "DB_PLC1_Send_To_PLC2_DB".CmdSeq := "DB_PLC1_Send_To_PLC2_DB".CmdSeq + 1;
   END_IF;
END_REGION

REGION Network 83: Handshake Client - Clear Latched Cmds on Ack
   RUNG wire#powerrail
      { S7_Templates := "SrcType := Int" } EQ_Contact(in1 := "DB_PLC1_Recv_From_PLC2_DB".AckSeq, in2 := "DB_PLC1_Send_To_PLC2_DB".CmdSeq)
      R_Coil( "DB_PLC1_Send_To_PLC2_DB".Cmd_Start )
   END_RUNG
   // the same network as SCL:
   IF "DB_PLC1_Recv_From_PLC2_DB".AckSeq = "DB_PLC1_Send_To_PLC2_DB".CmdSeq THEN
       "DB_PLC1_Send_To_PLC2_DB".Cmd_Start := FALSE;
   END_IF;
END_REGION

REGION Network 84: Handshake Client - Clear Latched Stop on Ack
   RUNG wire#powerrail
      { S7_Templates := "SrcType := Int" } EQ_Contact(in1 := "DB_PLC1_Recv_From_PLC2_DB".AckSeq, in2 := "DB_PLC1_Send_To_PLC2_DB".CmdSeq)
      R_Coil( "DB_PLC1_Send_To_PLC2_DB".Cmd_Stop )
   END_RUNG
   // the same network as SCL:
   IF "DB_PLC1_Recv_From_PLC2_DB".AckSeq = "DB_PLC1_Send_To_PLC2_DB".CmdSeq THEN
       "DB_PLC1_Send_To_PLC2_DB".Cmd_Stop := FALSE;
   END_IF;
END_REGION

REGION Network 85: Handshake Client - Clear Latched Reset on Ack
   RUNG wire#powerrail
      { S7_Templates := "SrcType := Int" } EQ_Contact(in1 := "DB_PLC1_Recv_From_PLC2_DB".AckSeq, in2 := "DB_PLC1_Send_To_PLC2_DB".CmdSeq)
      R_Coil( "DB_PLC1_Send_To_PLC2_DB".Cmd_Reset )
   END_RUNG
   // the same network as SCL:
   IF "DB_PLC1_Recv_From_PLC2_DB".AckSeq = "DB_PLC1_Send_To_PLC2_DB".CmdSeq THEN
       "DB_PLC1_Send_To_PLC2_DB".Cmd_Reset := FALSE;
   END_IF;
END_REGION

REGION Network 86: Handshake Client - Clear Latched EStop on Ack
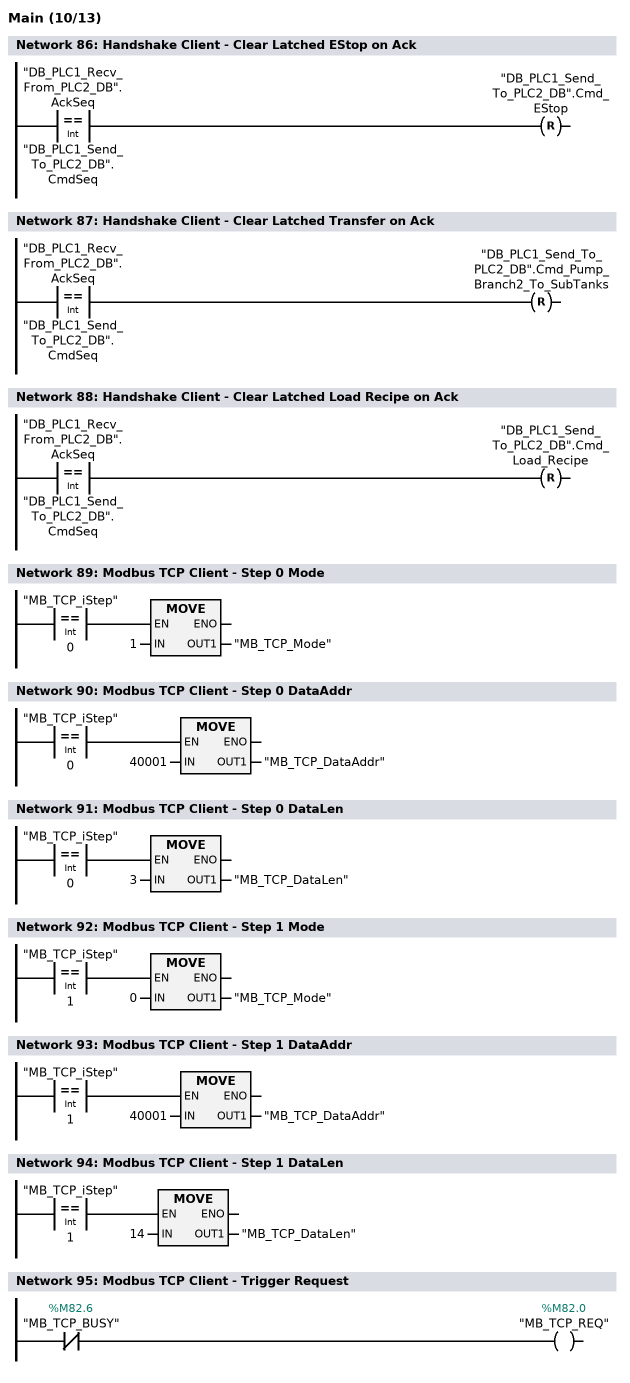
   RUNG wire#powerrail
      { S7_Templates := "SrcType := Int" } EQ_Contact(in1 := "DB_PLC1_Recv_From_PLC2_DB".AckSeq, in2 := "DB_PLC1_Send_To_PLC2_DB".CmdSeq)
      R_Coil( "DB_PLC1_Send_To_PLC2_DB".Cmd_EStop )
   END_RUNG
   // the same network as SCL:
   IF "DB_PLC1_Recv_From_PLC2_DB".AckSeq = "DB_PLC1_Send_To_PLC2_DB".CmdSeq THEN
       "DB_PLC1_Send_To_PLC2_DB".Cmd_EStop := FALSE;
   END_IF;
END_REGION

REGION Network 87: Handshake Client - Clear Latched Transfer on Ack
   RUNG wire#powerrail
      { S7_Templates := "SrcType := Int" } EQ_Contact(in1 := "DB_PLC1_Recv_From_PLC2_DB".AckSeq, in2 := "DB_PLC1_Send_To_PLC2_DB".CmdSeq)
      R_Coil( "DB_PLC1_Send_To_PLC2_DB".Cmd_Pump_Branch2_To_SubTanks )
   END_RUNG
   // the same network as SCL:
   IF "DB_PLC1_Recv_From_PLC2_DB".AckSeq = "DB_PLC1_Send_To_PLC2_DB".CmdSeq THEN
       "DB_PLC1_Send_To_PLC2_DB".Cmd_Pump_Branch2_To_SubTanks := FALSE;
   END_IF;
END_REGION

REGION Network 88: Handshake Client - Clear Latched Load Recipe on Ack
   RUNG wire#powerrail
      { S7_Templates := "SrcType := Int" } EQ_Contact(in1 := "DB_PLC1_Recv_From_PLC2_DB".AckSeq, in2 := "DB_PLC1_Send_To_PLC2_DB".CmdSeq)
      R_Coil( "DB_PLC1_Send_To_PLC2_DB".Cmd_Load_Recipe )
   END_RUNG
   // the same network as SCL:
   IF "DB_PLC1_Recv_From_PLC2_DB".AckSeq = "DB_PLC1_Send_To_PLC2_DB".CmdSeq THEN
       "DB_PLC1_Send_To_PLC2_DB".Cmd_Load_Recipe := FALSE;
   END_IF;
END_REGION

REGION Network 89: Modbus TCP Client - Step 0 Mode
   RUNG wire#powerrail
      { S7_Templates := "SrcType := Int" } EQ_Contact(in1 := "MB_TCP_iStep", in2 := 0)
      { S7_GenerateENO := "TRUE" } Move(in := 1, out1 => "MB_TCP_Mode")
   END_RUNG
   // the same network as SCL:
   IF "MB_TCP_iStep" = 0 THEN "MB_TCP_Mode" := 1; END_IF;
END_REGION

REGION Network 90: Modbus TCP Client - Step 0 DataAddr
   RUNG wire#powerrail
      { S7_Templates := "SrcType := Int" } EQ_Contact(in1 := "MB_TCP_iStep", in2 := 0)
      { S7_GenerateENO := "TRUE" } Move(in := 40001, out1 => "MB_TCP_DataAddr")
   END_RUNG
   // the same network as SCL:
   IF "MB_TCP_iStep" = 0 THEN "MB_TCP_DataAddr" := 40001; END_IF;
END_REGION

REGION Network 91: Modbus TCP Client - Step 0 DataLen
   RUNG wire#powerrail
      { S7_Templates := "SrcType := Int" } EQ_Contact(in1 := "MB_TCP_iStep", in2 := 0)
      { S7_GenerateENO := "TRUE" } Move(in := 3, out1 => "MB_TCP_DataLen")
   END_RUNG
   // the same network as SCL:
   IF "MB_TCP_iStep" = 0 THEN "MB_TCP_DataLen" := 3; END_IF;
END_REGION

REGION Network 92: Modbus TCP Client - Step 1 Mode
   RUNG wire#powerrail
      { S7_Templates := "SrcType := Int" } EQ_Contact(in1 := "MB_TCP_iStep", in2 := 1)
      { S7_GenerateENO := "TRUE" } Move(in := 0, out1 => "MB_TCP_Mode")
   END_RUNG
   // the same network as SCL:
   IF "MB_TCP_iStep" = 1 THEN "MB_TCP_Mode" := 0; END_IF;
END_REGION

REGION Network 93: Modbus TCP Client - Step 1 DataAddr
   RUNG wire#powerrail
      { S7_Templates := "SrcType := Int" } EQ_Contact(in1 := "MB_TCP_iStep", in2 := 1)
      { S7_GenerateENO := "TRUE" } Move(in := 40001, out1 => "MB_TCP_DataAddr")
   END_RUNG
   // the same network as SCL:
   IF "MB_TCP_iStep" = 1 THEN "MB_TCP_DataAddr" := 40001; END_IF;
END_REGION

REGION Network 94: Modbus TCP Client - Step 1 DataLen
   RUNG wire#powerrail
      { S7_Templates := "SrcType := Int" } EQ_Contact(in1 := "MB_TCP_iStep", in2 := 1)
      { S7_GenerateENO := "TRUE" } Move(in := 14, out1 => "MB_TCP_DataLen")
   END_RUNG
   // the same network as SCL:
   IF "MB_TCP_iStep" = 1 THEN "MB_TCP_DataLen" := 14; END_IF;
END_REGION

REGION Network 95: Modbus TCP Client - Trigger Request
   RUNG wire#powerrail
      I_Contact( "MB_TCP_BUSY" )
      Coil( "MB_TCP_REQ" )
   END_RUNG
   // the same network as SCL:
   "MB_TCP_REQ" := NOT "MB_TCP_BUSY";
END_REGION

REGION Network 96: Modbus TCP Client - Call MB_CLIENT
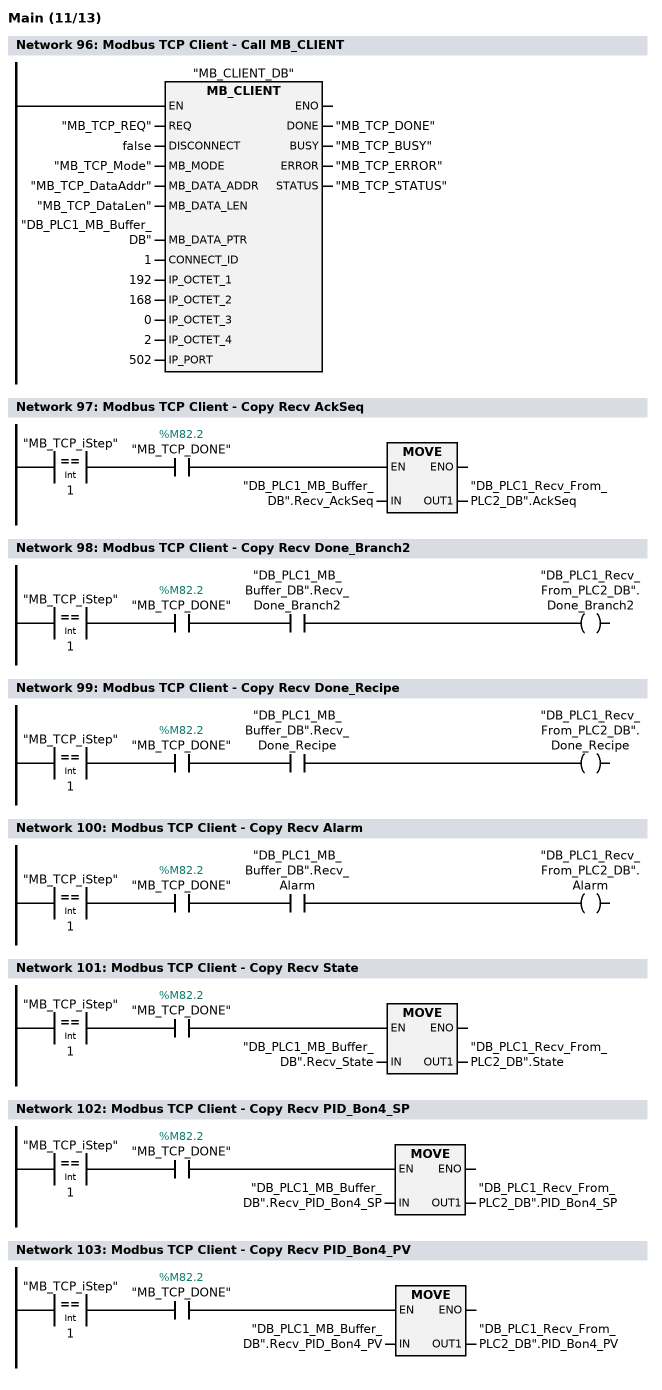
   RUNG wire#powerrail
      { S7_Templates := "[card1200 := 1, card1500 := 0]" } "MB_CLIENT_DB".MB_CLIENT(REQ := "MB_TCP_REQ", DISCONNECT := false, MB_MODE := "MB_TCP_Mode", MB_DATA_ADDR := "MB_TCP_DataAddr", MB_DATA_LEN := "MB_TCP_DataLen", MB_DATA_PTR := "DB_PLC1_MB_Buffer_DB", CONNECT_ID := 1, IP_OCTET_1 := 192, IP_OCTET_2 := 168, IP_OCTET_3 := 0, IP_OCTET_4 := 2, IP_PORT := 502, DONE => "MB_TCP_DONE", BUSY => "MB_TCP_BUSY", ERROR => "MB_TCP_ERROR", STATUS => "MB_TCP_STATUS")
   END_RUNG
   // the same network as SCL:
   "MB_CLIENT_DB"(REQ := "MB_TCP_REQ",   // MB_CLIENT
                  DISCONNECT := false,
                  MB_MODE := "MB_TCP_Mode",
                  MB_DATA_ADDR := "MB_TCP_DataAddr",
                  MB_DATA_LEN := "MB_TCP_DataLen",
                  MB_DATA_PTR := "DB_PLC1_MB_Buffer_DB",
                  CONNECT_ID := 1,
                  IP_OCTET_1 := 192,
                  IP_OCTET_2 := 168,
                  IP_OCTET_3 := 0,
                  IP_OCTET_4 := 2,
                  IP_PORT := 502,
                  DONE => "MB_TCP_DONE",
                  BUSY => "MB_TCP_BUSY",
                  ERROR => "MB_TCP_ERROR",
                  STATUS => "MB_TCP_STATUS");
END_REGION

REGION Network 97: Modbus TCP Client - Copy Recv AckSeq
   RUNG wire#powerrail
      { S7_Templates := "SrcType := Int" } EQ_Contact(in1 := "MB_TCP_iStep", in2 := 1)
      Contact( "MB_TCP_DONE" )
      { S7_GenerateENO := "TRUE" } Move(in := "DB_PLC1_MB_Buffer_DB".Recv_AckSeq, out1 => "DB_PLC1_Recv_From_PLC2_DB".AckSeq)
   END_RUNG
   // the same network as SCL:
   IF ("MB_TCP_iStep" = 1) AND "MB_TCP_DONE" THEN
       "DB_PLC1_Recv_From_PLC2_DB".AckSeq := "DB_PLC1_MB_Buffer_DB".Recv_AckSeq;
   END_IF;
END_REGION

REGION Network 98: Modbus TCP Client - Copy Recv Done_Branch2
   RUNG wire#powerrail
      { S7_Templates := "SrcType := Int" } EQ_Contact(in1 := "MB_TCP_iStep", in2 := 1)
      Contact( "MB_TCP_DONE" )
      Contact( "DB_PLC1_MB_Buffer_DB".Recv_Done_Branch2 )
      Coil( "DB_PLC1_Recv_From_PLC2_DB".Done_Branch2 )
   END_RUNG
   // the same network as SCL:
   "DB_PLC1_Recv_From_PLC2_DB".Done_Branch2 := ("MB_TCP_iStep" = 1) AND "MB_TCP_DONE" AND "DB_PLC1_MB_Buffer_DB".Recv_Done_Branch2;
END_REGION

REGION Network 99: Modbus TCP Client - Copy Recv Done_Recipe
   RUNG wire#powerrail
      { S7_Templates := "SrcType := Int" } EQ_Contact(in1 := "MB_TCP_iStep", in2 := 1)
      Contact( "MB_TCP_DONE" )
      Contact( "DB_PLC1_MB_Buffer_DB".Recv_Done_Recipe )
      Coil( "DB_PLC1_Recv_From_PLC2_DB".Done_Recipe )
   END_RUNG
   // the same network as SCL:
   "DB_PLC1_Recv_From_PLC2_DB".Done_Recipe := ("MB_TCP_iStep" = 1) AND "MB_TCP_DONE" AND "DB_PLC1_MB_Buffer_DB".Recv_Done_Recipe;
END_REGION

REGION Network 100: Modbus TCP Client - Copy Recv Alarm
   RUNG wire#powerrail
      { S7_Templates := "SrcType := Int" } EQ_Contact(in1 := "MB_TCP_iStep", in2 := 1)
      Contact( "MB_TCP_DONE" )
      Contact( "DB_PLC1_MB_Buffer_DB".Recv_Alarm )
      Coil( "DB_PLC1_Recv_From_PLC2_DB".Alarm )
   END_RUNG
   // the same network as SCL:
   "DB_PLC1_Recv_From_PLC2_DB".Alarm := ("MB_TCP_iStep" = 1) AND "MB_TCP_DONE" AND "DB_PLC1_MB_Buffer_DB".Recv_Alarm;
END_REGION

REGION Network 101: Modbus TCP Client - Copy Recv State
   RUNG wire#powerrail
      { S7_Templates := "SrcType := Int" } EQ_Contact(in1 := "MB_TCP_iStep", in2 := 1)
      Contact( "MB_TCP_DONE" )
      { S7_GenerateENO := "TRUE" } Move(in := "DB_PLC1_MB_Buffer_DB".Recv_State, out1 => "DB_PLC1_Recv_From_PLC2_DB".State)
   END_RUNG
   // the same network as SCL:
   IF ("MB_TCP_iStep" = 1) AND "MB_TCP_DONE" THEN
       "DB_PLC1_Recv_From_PLC2_DB".State := "DB_PLC1_MB_Buffer_DB".Recv_State;
   END_IF;
END_REGION

REGION Network 102: Modbus TCP Client - Copy Recv PID_Bon4_SP
   RUNG wire#powerrail
      { S7_Templates := "SrcType := Int" } EQ_Contact(in1 := "MB_TCP_iStep", in2 := 1)
      Contact( "MB_TCP_DONE" )
      { S7_GenerateENO := "TRUE" } Move(in := "DB_PLC1_MB_Buffer_DB".Recv_PID_Bon4_SP, out1 => "DB_PLC1_Recv_From_PLC2_DB".PID_Bon4_SP)
   END_RUNG
   // the same network as SCL:
   IF ("MB_TCP_iStep" = 1) AND "MB_TCP_DONE" THEN
       "DB_PLC1_Recv_From_PLC2_DB".PID_Bon4_SP := "DB_PLC1_MB_Buffer_DB".Recv_PID_Bon4_SP;
   END_IF;
END_REGION

REGION Network 103: Modbus TCP Client - Copy Recv PID_Bon4_PV
   RUNG wire#powerrail
      { S7_Templates := "SrcType := Int" } EQ_Contact(in1 := "MB_TCP_iStep", in2 := 1)
      Contact( "MB_TCP_DONE" )
      { S7_GenerateENO := "TRUE" } Move(in := "DB_PLC1_MB_Buffer_DB".Recv_PID_Bon4_PV, out1 => "DB_PLC1_Recv_From_PLC2_DB".PID_Bon4_PV)
   END_RUNG
   // the same network as SCL:
   IF ("MB_TCP_iStep" = 1) AND "MB_TCP_DONE" THEN
       "DB_PLC1_Recv_From_PLC2_DB".PID_Bon4_PV := "DB_PLC1_MB_Buffer_DB".Recv_PID_Bon4_PV;
   END_IF;
END_REGION

REGION Network 104: Modbus TCP Client - Copy Recv PID_Bon4_CV
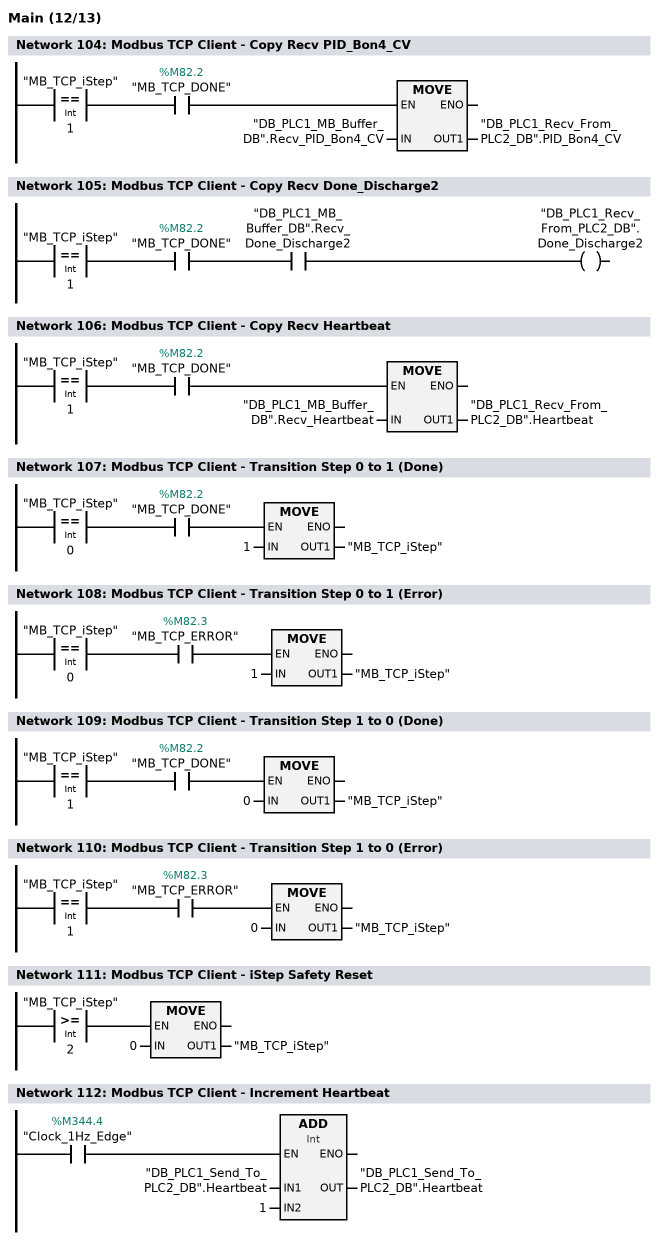
   RUNG wire#powerrail
      { S7_Templates := "SrcType := Int" } EQ_Contact(in1 := "MB_TCP_iStep", in2 := 1)
      Contact( "MB_TCP_DONE" )
      { S7_GenerateENO := "TRUE" } Move(in := "DB_PLC1_MB_Buffer_DB".Recv_PID_Bon4_CV, out1 => "DB_PLC1_Recv_From_PLC2_DB".PID_Bon4_CV)
   END_RUNG
   // the same network as SCL:
   IF ("MB_TCP_iStep" = 1) AND "MB_TCP_DONE" THEN
       "DB_PLC1_Recv_From_PLC2_DB".PID_Bon4_CV := "DB_PLC1_MB_Buffer_DB".Recv_PID_Bon4_CV;
   END_IF;
END_REGION

REGION Network 105: Modbus TCP Client - Copy Recv Done_Discharge2
   RUNG wire#powerrail
      { S7_Templates := "SrcType := Int" } EQ_Contact(in1 := "MB_TCP_iStep", in2 := 1)
      Contact( "MB_TCP_DONE" )
      Contact( "DB_PLC1_MB_Buffer_DB".Recv_Done_Discharge2 )
      Coil( "DB_PLC1_Recv_From_PLC2_DB".Done_Discharge2 )
   END_RUNG
   // the same network as SCL:
   "DB_PLC1_Recv_From_PLC2_DB".Done_Discharge2 := ("MB_TCP_iStep" = 1) AND "MB_TCP_DONE" AND "DB_PLC1_MB_Buffer_DB".Recv_Done_Discharge2;
END_REGION

REGION Network 106: Modbus TCP Client - Copy Recv Heartbeat
   RUNG wire#powerrail
      { S7_Templates := "SrcType := Int" } EQ_Contact(in1 := "MB_TCP_iStep", in2 := 1)
      Contact( "MB_TCP_DONE" )
      { S7_GenerateENO := "TRUE" } Move(in := "DB_PLC1_MB_Buffer_DB".Recv_Heartbeat, out1 => "DB_PLC1_Recv_From_PLC2_DB".Heartbeat)
   END_RUNG
   // the same network as SCL:
   IF ("MB_TCP_iStep" = 1) AND "MB_TCP_DONE" THEN
       "DB_PLC1_Recv_From_PLC2_DB".Heartbeat := "DB_PLC1_MB_Buffer_DB".Recv_Heartbeat;
   END_IF;
END_REGION

REGION Network 107: Modbus TCP Client - Transition Step 0 to 1 (Done)
   RUNG wire#powerrail
      { S7_Templates := "SrcType := Int" } EQ_Contact(in1 := "MB_TCP_iStep", in2 := 0)
      Contact( "MB_TCP_DONE" )
      { S7_GenerateENO := "TRUE" } Move(in := 1, out1 => "MB_TCP_iStep")
   END_RUNG
   // the same network as SCL:
   IF ("MB_TCP_iStep" = 0) AND "MB_TCP_DONE" THEN "MB_TCP_iStep" := 1; END_IF;
END_REGION

REGION Network 108: Modbus TCP Client - Transition Step 0 to 1 (Error)
   RUNG wire#powerrail
      { S7_Templates := "SrcType := Int" } EQ_Contact(in1 := "MB_TCP_iStep", in2 := 0)
      Contact( "MB_TCP_ERROR" )
      { S7_GenerateENO := "TRUE" } Move(in := 1, out1 => "MB_TCP_iStep")
   END_RUNG
   // the same network as SCL:
   IF ("MB_TCP_iStep" = 0) AND "MB_TCP_ERROR" THEN "MB_TCP_iStep" := 1; END_IF;
END_REGION

REGION Network 109: Modbus TCP Client - Transition Step 1 to 0 (Done)
   RUNG wire#powerrail
      { S7_Templates := "SrcType := Int" } EQ_Contact(in1 := "MB_TCP_iStep", in2 := 1)
      Contact( "MB_TCP_DONE" )
      { S7_GenerateENO := "TRUE" } Move(in := 0, out1 => "MB_TCP_iStep")
   END_RUNG
   // the same network as SCL:
   IF ("MB_TCP_iStep" = 1) AND "MB_TCP_DONE" THEN "MB_TCP_iStep" := 0; END_IF;
END_REGION

REGION Network 110: Modbus TCP Client - Transition Step 1 to 0 (Error)
   RUNG wire#powerrail
      { S7_Templates := "SrcType := Int" } EQ_Contact(in1 := "MB_TCP_iStep", in2 := 1)
      Contact( "MB_TCP_ERROR" )
      { S7_GenerateENO := "TRUE" } Move(in := 0, out1 => "MB_TCP_iStep")
   END_RUNG
   // the same network as SCL:
   IF ("MB_TCP_iStep" = 1) AND "MB_TCP_ERROR" THEN "MB_TCP_iStep" := 0; END_IF;
END_REGION

REGION Network 111: Modbus TCP Client - iStep Safety Reset
   RUNG wire#powerrail
      { S7_Templates := "SrcType := Int" } GE_Contact(in1 := "MB_TCP_iStep", in2 := 2)
      { S7_GenerateENO := "TRUE" } Move(in := 0, out1 => "MB_TCP_iStep")
   END_RUNG
   // the same network as SCL:
   IF "MB_TCP_iStep" >= 2 THEN "MB_TCP_iStep" := 0; END_IF;
END_REGION

REGION Network 112: Modbus TCP Client - Increment Heartbeat
   RUNG wire#powerrail
      Contact( "Clock_1Hz_Edge" )
      { S7_Templates := "SrcType := Int"; S7_GenerateENO := "TRUE" } Add(in1 := "DB_PLC1_Send_To_PLC2_DB".Heartbeat, in2 := 1, out => "DB_PLC1_Send_To_PLC2_DB".Heartbeat)
   END_RUNG
   // the same network as SCL:
   IF "Clock_1Hz_Edge" THEN
       "DB_PLC1_Send_To_PLC2_DB".Heartbeat := "DB_PLC1_Send_To_PLC2_DB".Heartbeat + 1;
   END_IF;
END_REGION

REGION Network 113: Modbus TCP Client - Monitor Heartbeat Change
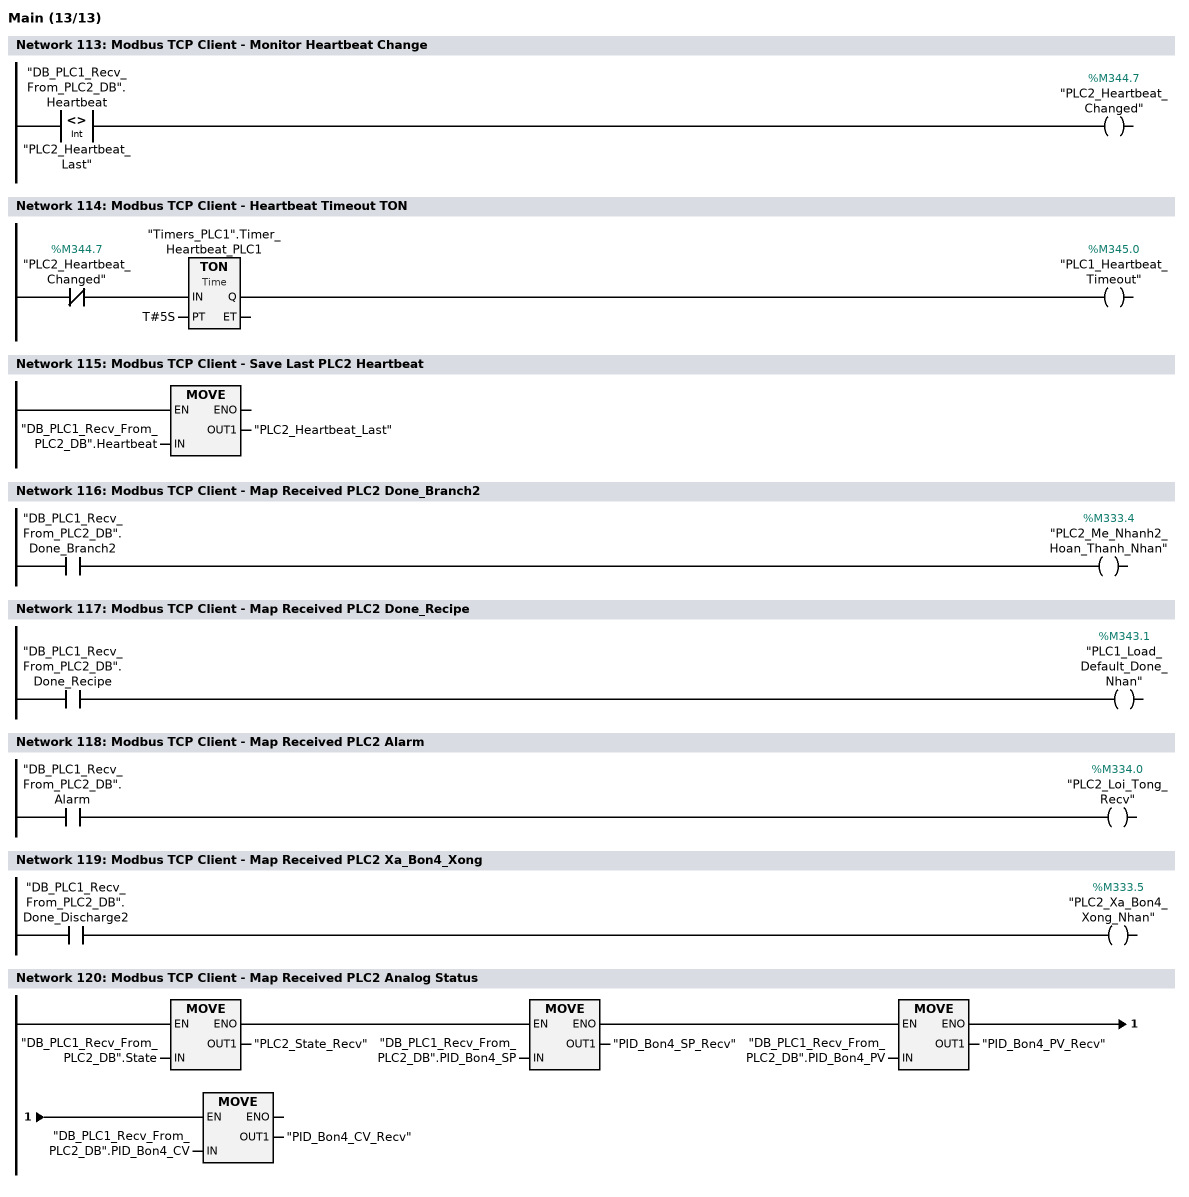
   RUNG wire#powerrail
      { S7_Templates := "SrcType := Int" } NE_Contact(in1 := "DB_PLC1_Recv_From_PLC2_DB".Heartbeat, in2 := "PLC2_Heartbeat_Last")
      Coil( "PLC2_Heartbeat_Changed" )
   END_RUNG
   // the same network as SCL:
   "PLC2_Heartbeat_Changed" := "DB_PLC1_Recv_From_PLC2_DB".Heartbeat <> "PLC2_Heartbeat_Last";
END_REGION

REGION Network 114: Modbus TCP Client - Heartbeat Timeout TON
   RUNG wire#powerrail
      I_Contact( "PLC2_Heartbeat_Changed" )
      { S7_Templates := "time_type := Time" } "Timers_PLC1".Timer_Heartbeat_PLC1.TON(pt := T#5S, et =>)
      Coil( "PLC1_Heartbeat_Timeout" )
   END_RUNG
   // the same network as SCL:
   "Timers_PLC1".Timer_Heartbeat_PLC1.TON(IN := NOT "PLC2_Heartbeat_Changed", PT := T#5S);
   "PLC1_Heartbeat_Timeout" := "Timers_PLC1".Timer_Heartbeat_PLC1.Q;
END_REGION

REGION Network 115: Modbus TCP Client - Save Last PLC2 Heartbeat
   RUNG wire#powerrail
      { S7_GenerateENO := "TRUE" } Move(in := "DB_PLC1_Recv_From_PLC2_DB".Heartbeat, out1 => "PLC2_Heartbeat_Last")
   END_RUNG
   // the same network as SCL:
   "PLC2_Heartbeat_Last" := "DB_PLC1_Recv_From_PLC2_DB".Heartbeat;
END_REGION

REGION Network 116: Modbus TCP Client - Map Received PLC2 Done_Branch2
   RUNG wire#powerrail
      Contact( "DB_PLC1_Recv_From_PLC2_DB".Done_Branch2 )
      Coil( "PLC2_Me_Nhanh2_Hoan_Thanh_Nhan" )
   END_RUNG
   // the same network as SCL:
   "PLC2_Me_Nhanh2_Hoan_Thanh_Nhan" := "DB_PLC1_Recv_From_PLC2_DB".Done_Branch2;
END_REGION

REGION Network 117: Modbus TCP Client - Map Received PLC2 Done_Recipe
   RUNG wire#powerrail
      Contact( "DB_PLC1_Recv_From_PLC2_DB".Done_Recipe )
      Coil( "PLC1_Load_Default_Done_Nhan" )
   END_RUNG
   // the same network as SCL:
   "PLC1_Load_Default_Done_Nhan" := "DB_PLC1_Recv_From_PLC2_DB".Done_Recipe;
END_REGION

REGION Network 118: Modbus TCP Client - Map Received PLC2 Alarm
   RUNG wire#powerrail
      Contact( "DB_PLC1_Recv_From_PLC2_DB".Alarm )
      Coil( "PLC2_Loi_Tong_Recv" )
   END_RUNG
   // the same network as SCL:
   "PLC2_Loi_Tong_Recv" := "DB_PLC1_Recv_From_PLC2_DB".Alarm;
END_REGION

REGION Network 119: Modbus TCP Client - Map Received PLC2 Xa_Bon4_Xong
   RUNG wire#powerrail
      Contact( "DB_PLC1_Recv_From_PLC2_DB".Done_Discharge2 )
      Coil( "PLC2_Xa_Bon4_Xong_Nhan" )
   END_RUNG
   // the same network as SCL:
   "PLC2_Xa_Bon4_Xong_Nhan" := "DB_PLC1_Recv_From_PLC2_DB".Done_Discharge2;
END_REGION

REGION Network 120: Modbus TCP Client - Map Received PLC2 Analog Status
   RUNG wire#powerrail
      { S7_GenerateENO := "TRUE" } Move(in := "DB_PLC1_Recv_From_PLC2_DB".State, out1 => "PLC2_State_Recv")
      { S7_GenerateENO := "TRUE" } Move(in := "DB_PLC1_Recv_From_PLC2_DB".PID_Bon4_SP, out1 => "PID_Bon4_SP_Recv")
      { S7_GenerateENO := "TRUE" } Move(in := "DB_PLC1_Recv_From_PLC2_DB".PID_Bon4_PV, out1 => "PID_Bon4_PV_Recv")
      { S7_GenerateENO := "TRUE" } Move(in := "DB_PLC1_Recv_From_PLC2_DB".PID_Bon4_CV, out1 => "PID_Bon4_CV_Recv")
   END_RUNG
   // the same network as SCL:
   // ENO of a box is taken as its EN; it also drops when the box reports an error
   "PLC2_State_Recv" := "DB_PLC1_Recv_From_PLC2_DB".State;
   "PID_Bon4_SP_Recv" := "DB_PLC1_Recv_From_PLC2_DB".PID_Bon4_SP;
   "PID_Bon4_PV_Recv" := "DB_PLC1_Recv_From_PLC2_DB".PID_Bon4_PV;
   "PID_Bon4_CV_Recv" := "DB_PLC1_Recv_From_PLC2_DB".PID_Bon4_CV;
END_REGION
END_ORGANIZATION_BLOCK

FUNCTION "FC_Init_Default_Recipe_PLC1" : Void   // FC50, LAD
{ S7_Optimized_Access := 'TRUE' }
VERSION : 0.1
// stored: AutoNumber true, IsIECCheckEnabled false, SetENOAutomatically false, UDAEnableTagReadback false
BEGIN

REGION Network 1: Kích hoạt nạp recipe mặc định lần đầu scan PLC1
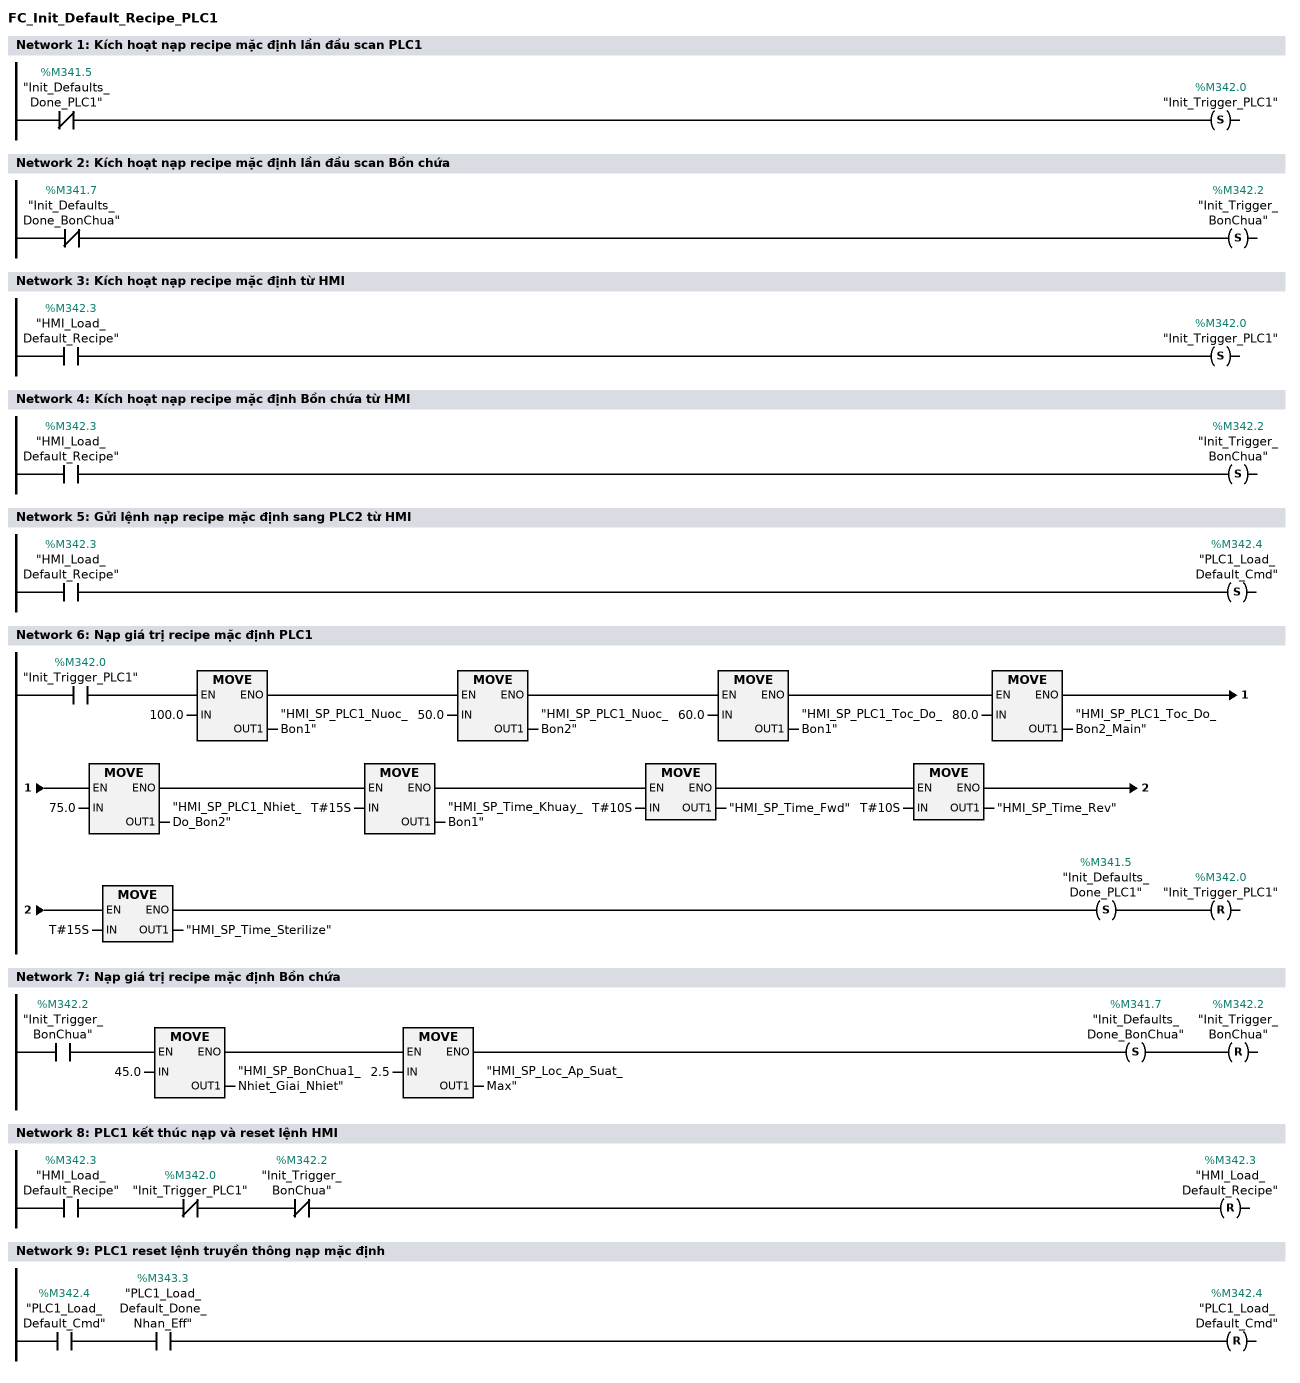
   RUNG wire#powerrail
      I_Contact( "Init_Defaults_Done_PLC1" )
      S_Coil( "Init_Trigger_PLC1" )
   END_RUNG
   // the same network as SCL:
   IF NOT "Init_Defaults_Done_PLC1" THEN "Init_Trigger_PLC1" := TRUE; END_IF;
END_REGION

REGION Network 2: Kích hoạt nạp recipe mặc định lần đầu scan Bồn chứa
   RUNG wire#powerrail
      I_Contact( "Init_Defaults_Done_BonChua" )
      S_Coil( "Init_Trigger_BonChua" )
   END_RUNG
   // the same network as SCL:
   IF NOT "Init_Defaults_Done_BonChua" THEN "Init_Trigger_BonChua" := TRUE; END_IF;
END_REGION

REGION Network 3: Kích hoạt nạp recipe mặc định từ HMI
   RUNG wire#powerrail
      Contact( "HMI_Load_Default_Recipe" )
      S_Coil( "Init_Trigger_PLC1" )
   END_RUNG
   // the same network as SCL:
   IF "HMI_Load_Default_Recipe" THEN "Init_Trigger_PLC1" := TRUE; END_IF;
END_REGION

REGION Network 4: Kích hoạt nạp recipe mặc định Bồn chứa từ HMI
   RUNG wire#powerrail
      Contact( "HMI_Load_Default_Recipe" )
      S_Coil( "Init_Trigger_BonChua" )
   END_RUNG
   // the same network as SCL:
   IF "HMI_Load_Default_Recipe" THEN "Init_Trigger_BonChua" := TRUE; END_IF;
END_REGION

REGION Network 5: Gửi lệnh nạp recipe mặc định sang PLC2 từ HMI
   RUNG wire#powerrail
      Contact( "HMI_Load_Default_Recipe" )
      S_Coil( "PLC1_Load_Default_Cmd" )
   END_RUNG
   // the same network as SCL:
   IF "HMI_Load_Default_Recipe" THEN "PLC1_Load_Default_Cmd" := TRUE; END_IF;
END_REGION

REGION Network 6: Nạp giá trị recipe mặc định PLC1
   RUNG wire#powerrail
      Contact( "Init_Trigger_PLC1" )
      { S7_GenerateENO := "TRUE" } Move(in := 100.0, out1 => "HMI_SP_PLC1_Nuoc_Bon1")
      { S7_GenerateENO := "TRUE" } Move(in := 50.0, out1 => "HMI_SP_PLC1_Nuoc_Bon2")
      { S7_GenerateENO := "TRUE" } Move(in := 60.0, out1 => "HMI_SP_PLC1_Toc_Do_Bon1")
      { S7_GenerateENO := "TRUE" } Move(in := 80.0, out1 => "HMI_SP_PLC1_Toc_Do_Bon2_Main")
      { S7_GenerateENO := "TRUE" } Move(in := 75.0, out1 => "HMI_SP_PLC1_Nhiet_Do_Bon2")
      { S7_GenerateENO := "TRUE" } Move(in := T#15S, out1 => "HMI_SP_Time_Khuay_Bon1")
      { S7_GenerateENO := "TRUE" } Move(in := T#10S, out1 => "HMI_SP_Time_Fwd")
      { S7_GenerateENO := "TRUE" } Move(in := T#10S, out1 => "HMI_SP_Time_Rev")
      { S7_GenerateENO := "TRUE" } Move(in := T#15S, out1 => "HMI_SP_Time_Sterilize")
      S_Coil( "Init_Defaults_Done_PLC1" )
      R_Coil( "Init_Trigger_PLC1" )
   END_RUNG
   // the same network as SCL:
   // ENO of a box is taken as its EN; it also drops when the box reports an error
   IF "Init_Trigger_PLC1" THEN
       "HMI_SP_PLC1_Nuoc_Bon1" := 100.0;
       "HMI_SP_PLC1_Nuoc_Bon2" := 50.0;
       "HMI_SP_PLC1_Toc_Do_Bon1" := 60.0;
       "HMI_SP_PLC1_Toc_Do_Bon2_Main" := 80.0;
       "HMI_SP_PLC1_Nhiet_Do_Bon2" := 75.0;
       "HMI_SP_Time_Khuay_Bon1" := T#15S;
       "HMI_SP_Time_Fwd" := T#10S;
       "HMI_SP_Time_Rev" := T#10S;
       "HMI_SP_Time_Sterilize" := T#15S;
       "Init_Defaults_Done_PLC1" := TRUE;
       "Init_Trigger_PLC1" := FALSE;
   END_IF;
END_REGION

REGION Network 7: Nạp giá trị recipe mặc định Bồn chứa
   RUNG wire#powerrail
      Contact( "Init_Trigger_BonChua" )
      { S7_GenerateENO := "TRUE" } Move(in := 45.0, out1 => "HMI_SP_BonChua1_Nhiet_Giai_Nhiet")
      { S7_GenerateENO := "TRUE" } Move(in := 2.5, out1 => "HMI_SP_Loc_Ap_Suat_Max")
      S_Coil( "Init_Defaults_Done_BonChua" )
      R_Coil( "Init_Trigger_BonChua" )
   END_RUNG
   // the same network as SCL:
   // ENO of a box is taken as its EN; it also drops when the box reports an error
   IF "Init_Trigger_BonChua" THEN
       "HMI_SP_BonChua1_Nhiet_Giai_Nhiet" := 45.0;
       "HMI_SP_Loc_Ap_Suat_Max" := 2.5;
       "Init_Defaults_Done_BonChua" := TRUE;
       "Init_Trigger_BonChua" := FALSE;
   END_IF;
END_REGION

REGION Network 8: PLC1 kết thúc nạp và reset lệnh HMI
   RUNG wire#powerrail
      Contact( "HMI_Load_Default_Recipe" )
      I_Contact( "Init_Trigger_PLC1" )
      I_Contact( "Init_Trigger_BonChua" )
      R_Coil( "HMI_Load_Default_Recipe" )
   END_RUNG
   // the same network as SCL:
   IF "HMI_Load_Default_Recipe" AND NOT "Init_Trigger_PLC1" AND NOT "Init_Trigger_BonChua" THEN
       "HMI_Load_Default_Recipe" := FALSE;
   END_IF;
END_REGION

REGION Network 9: PLC1 reset lệnh truyền thông nạp mặc định
   RUNG wire#powerrail
      Contact( "PLC1_Load_Default_Cmd" )
      Contact( "PLC1_Load_Default_Done_Nhan_Eff" )
      R_Coil( "PLC1_Load_Default_Cmd" )
   END_RUNG
   // the same network as SCL:
   IF "PLC1_Load_Default_Cmd" AND "PLC1_Load_Default_Done_Nhan_Eff" THEN
       "PLC1_Load_Default_Cmd" := FALSE;
   END_IF;
END_REGION
END_FUNCTION

